KUKA KRL program: MyProgram_288().src

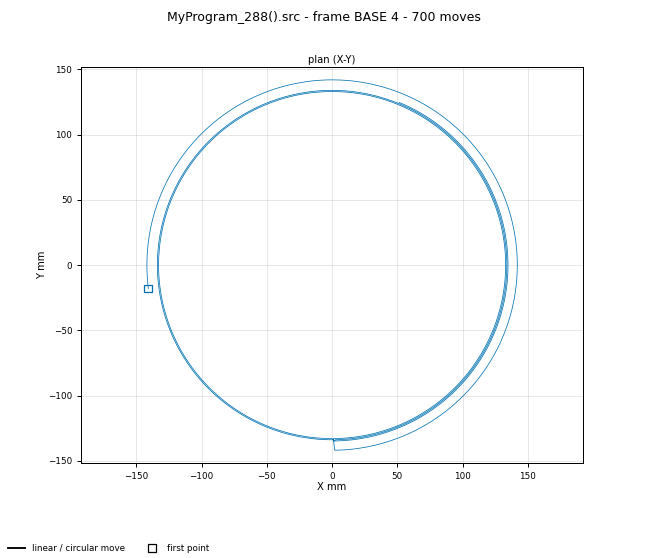
[picture p0: tool path of MyProgram_288().src in frame BASE 4, 700 of 700 moves have a stored position in this frame; points joined in program order, loops and branches not executed]
&ACCESS RVP
&REL 1
&PARAM TEMPLATE = C:\KRC\Roboter\Template\vorgabe
&PARAM EDITMASK = *
DEF MyProgram_288()
; ---- Setting reference (Base) ----
$BASE = BASE_DATA[4]

; --------------------------
; ---- Setting tool (TCP) ----
$TOOL = TOOL_DATA[3]
; --------------------------

$VEL.CP = VEL_APROX_PRINT
Startdeposition()
$VEL.CP = VEL_PRINT
LIN {X -140.7234,Y -17.946,Z 175,A -170.729,B 7.332,C 0.3003,E1 7.1791,E2 262.9088} C_DIS
LIN {X -141.1414,Y -14.3037,Z 175,A -172.2619,B 7.332,C 0.2967,E1 7.1786,E2 264.4473} C_DIS
LIN {X -141.4779,Y -10.4373,Z 175,A -173.8413,B 7.3323,C 0.2924,E1 7.1783,E2 266.0269} C_DIS
LIN {X -141.6907,Y -6.9788,Z 175,A -175.2622,B 7.3324,C 0.2887,E1 7.178,E2 267.4494} C_DIS
LIN {X -141.8124,Y -3.7701,Z 175,A -176.5843,B 7.3326,C 0.2853,E1 7.178,E2 268.7736} C_DIS
LIN {X -141.8652,Y -0.0247,Z 175,A -178.1224,B 7.3327,C 0.2813,E1 7.1779,E2 270.3138} C_DIS
LIN {X -141.8205,Y 3.4801,Z 175,A -179.5927,B 7.3328,C 0.2779,E1 7.1779,E2 271.7898} C_DIS
LIN {X -141.7054,Y 6.6857,Z 175,A 179.0865,B 7.333,C 0.2746,E1 7.1781,E2 273.1128} C_DIS
LIN {X -141.499,Y 10.1492,Z 175,A 177.6636,B 7.333,C 0.2708,E1 7.1784,E2 274.5373} C_DIS
LIN {X -141.1833,Y 13.8665,Z 175,A 176.1372,B 7.3332,C 0.2668,E1 7.1788,E2 276.0648} C_DIS
LIN {X -140.7964,Y 17.3669,Z 175,A 174.6904,B 7.3334,C 0.263,E1 7.1792,E2 277.5136} C_DIS
LIN {X -140.3316,Y 20.7961,Z 175,A 173.2648,B 7.3335,C 0.2594,E1 7.1798,E2 278.9414} C_DIS
LIN {X -139.825,Y 23.9636,Z 175,A 171.9397,B 7.3336,C 0.2561,E1 7.1804,E2 280.2692} C_DIS
LIN {X -139.1474,Y 27.6283,Z 175,A 170.388,B 7.3337,C 0.2525,E1 7.1812,E2 281.8255} C_DIS
LIN {X -138.5463,Y 30.4976,Z 175,A 169.1448,B 7.3338,C 0.2499,E1 7.1819,E2 283.0752} C_DIS
LIN {X -137.6088,Y 34.4796,Z 175,A 167.4991,B 7.334,C 0.2452,E1 7.183,E2 284.7185} C_DIS
LIN {X -136.7221,Y 37.8424,Z 175,A 166.1483,B 7.3341,C 0.2406,E1 7.184,E2 286.061} C_DIS
LIN {X -135.8307,Y 40.9296,Z 175,A 164.745,B 7.3342,C 0.2384,E1 7.1851,E2 287.4766} C_DIS
LIN {X -134.7033,Y 44.4966,Z 175,A 163.206,B 7.3343,C 0.2346,E1 7.1864,E2 289.0178} C_DIS
LIN {X -133.6609,Y 47.5391,Z 175,A 161.8116,B 7.3344,C 0.2324,E1 7.1877,E2 290.4232} C_DIS
LIN {X -132.3609,Y 51.0445,Z 175,A 160.4261,B 7.3346,C 0.2266,E1 7.1891,E2 291.7913} C_DIS
LIN {X -131.2247,Y 53.9034,Z 175,A 159.0704,B 7.3346,C 0.2248,E1 7.1905,E2 293.1604} C_DIS
LIN {X -129.8606,Y 57.112,Z 175,A 157.5842,B 7.3347,C 0.2221,E1 7.1922,E2 294.6552} C_DIS
LIN {X -128.3684,Y 60.3909,Z 175,A 156.1693,B 7.3349,C 0.2178,E1 7.1938,E2 296.0636} C_DIS
LIN {X -127.1018,Y 63.008,Z 175,A 154.9452,B 7.3349,C 0.2154,E1 7.1953,E2 297.2929} C_DIS
LIN {X -125.1762,Y 66.7568,Z 175,A 153.2018,B 7.335,C 0.2116,E1 7.1976,E2 299.04} C_DIS
LIN {X -123.1184,Y 70.4789,Z 175,A 151.466,B 7.3351,C 0.2075,E1 7.2,E2 300.7764} C_DIS
LIN {X -121.2352,Y 73.6715,Z 175,A 149.9398,B 7.3352,C 0.2042,E1 7.2021,E2 302.3049} C_DIS
LIN {X -118.9968,Y 77.2342,Z 175,A 148.2034,B 7.3353,C 0.2006,E1 7.2048,E2 304.0443} C_DIS
LIN {X -117.0516,Y 80.1517,Z 175,A 146.7407,B 7.3354,C 0.1978,E1 7.207,E2 305.5116} C_DIS
LIN {X -114.4633,Y 83.8067,Z 175,A 144.8252,B 7.3354,C 0.195,E1 7.2102,E2 307.439} C_DIS
LIN {X -111.8255,Y 87.2959,Z 175,A 143.1344,B 7.3356,C 0.1899,E1 7.213,E2 309.1185} C_DIS
LIN {X -109.1286,Y 90.6441,Z 175,A 141.2584,B 7.3356,C 0.188,E1 7.2164,E2 311.0106} C_DIS
LIN {X -106.2303,Y 94.0238,Z 175,A 139.4357,B 7.3358,C 0.1844,E1 7.2197,E2 312.8347} C_DIS
LIN {X -102.8784,Y 97.6811,Z 175,A 137.4601,B 7.3358,C 0.1798,E1 7.2235,E2 314.8049} C_DIS
LIN {X -99.7959,Y 100.8276,Z 175,A 135.6913,B 7.336,C 0.176,E1 7.227,E2 316.5708} C_DIS
LIN {X -96.667,Y 103.8308,Z 175,A 133.9289,B 7.336,C 0.1726,E1 7.2305,E2 318.3329} C_DIS
LIN {X -93.4431,Y 106.7417,Z 175,A 132.149,B 7.3361,C 0.1696,E1 7.2342,E2 320.1146} C_DIS
LIN {X -90.672,Y 109.1055,Z 175,A 130.5573,B 7.3361,C 0.1686,E1 7.2377,E2 321.7203} C_DIS
LIN {X -87.4029,Y 111.7415,Z 175,A 128.9292,B 7.3362,C 0.1646,E1 7.2412,E2 323.3382} C_DIS
LIN {X -83.8422,Y 114.4372,Z 175,A 127.0041,B 7.3362,C 0.1632,E1 7.2456,E2 325.2771} C_DIS
LIN {X -80.1816,Y 117.0311,Z 175,A 125.1904,B 7.3363,C 0.1603,E1 7.2497,E2 327.0895} C_DIS
LIN {X -76.6264,Y 119.3892,Z 175,A 123.4418,B 7.3363,C 0.1579,E1 7.2538,E2 328.8399} C_DIS
LIN {X -72.8225,Y 121.7468,Z 175,A 121.6324,B 7.3364,C 0.1553,E1 7.2581,E2 330.648} C_DIS
LIN {X -69.0599,Y 123.9203,Z 175,A 119.8443,B 7.3364,C 0.1532,E1 7.2625,E2 332.439} C_DIS
LIN {X -65.3363,Y 125.9223,Z 175,A 118.2406,B 7.3366,C 0.1494,E1 7.2664,E2 334.0281} C_DIS
LIN {X -62.3478,Y 127.4274,Z 175,A 116.9025,B 7.3366,C 0.1475,E1 7.2697,E2 335.3635} C_DIS
LIN {X -59.0667,Y 128.9814,Z 175,A 115.3957,B 7.3366,C 0.1463,E1 7.2736,E2 336.8742} C_DIS
LIN {X -55.8949,Y 130.3869,Z 175,A 113.9847,B 7.3366,C 0.1448,E1 7.2772,E2 338.2854} C_DIS
LIN {X -52.6901,Y 131.7145,Z 175,A 112.5741,B 7.3366,C 0.1434,E1 7.2808,E2 339.6962} C_DIS
LIN {X -49.6954,Y 132.8728,Z 175,A 111.2695,B 7.3366,C 0.1422,E1 7.2842,E2 341.0008} C_DIS
LIN {X -46.1824,Y 134.1346,Z 175,A 109.8377,B 7.3367,C 0.1396,E1 7.288,E2 342.422} C_DIS
LIN {X -43.0961,Y 135.1575,Z 175,A 108.3928,B 7.3367,C 0.1405,E1 7.2919,E2 343.8827} C_DIS
LIN {X -39.5162,Y 136.2477,Z 175,A 106.9116,B 7.3367,C 0.1388,E1 7.2958,E2 345.3591} C_DIS
LIN {X -36.4172,Y 137.1082,Z 175,A 105.7185,B 7.3368,C 0.1362,E1 7.299,E2 346.5378} C_DIS
LIN {X -33.032,Y 137.963,Z 175,A 104.1617,B 7.3368,C 0.1375,E1 7.3033,E2 348.1124} C_DIS
LIN {X -29.4095,Y 138.7812,Z 175,A 102.7067,B 7.3368,C 0.1359,E1 7.3072,E2 349.5608} C_DIS
LIN {X -26.2675,Y 139.4096,Z 175,A 101.3667,B 7.3368,C 0.1359,E1 7.3109,E2 350.9058} C_DIS
LIN {X -22.5864,Y 140.0547,Z 175,A 99.8841,B 7.3368,C 0.1347,E1 7.315,E2 352.3841} C_DIS
LIN {X -19.3533,Y 140.5378,Z 175,A 98.557,B 7.3368,C 0.1343,E1 7.3186,E2 353.7114} C_DIS
LIN {X -15.9024,Y 140.97,Z 175,A 97.1856,B 7.3368,C 0.1333,E1 7.3224,E2 355.0778} C_DIS
LIN {X -12.4434,Y 141.3164,Z 175,A 95.6611,B 7.3368,C 0.1348,E1 7.3267,E2 356.6168} C_DIS
LIN {X -8.7043,Y 141.5951,Z 175,A 94.091,B 7.3368,C 0.1354,E1 7.3311,E2 358.1931} C_DIS
LIN {X -3.7458,Y 141.8131,Z 175,A 92.2151,B 7.3368,C 0.1332,E1 7.3363,E2 360.0518} C_DIS
LIN {X -0.0049,Y 141.8646,Z 175,A 90.7261,B 7.3368,C 0.1328,E1 7.3404,E2 361.5374} C_DIS
LIN {X 3.4708,Y 141.8207,Z 175,A 89.2787,B 7.3368,C 0.1336,E1 7.3445,E2 362.9897} C_DIS
LIN {X 6.6856,Y 141.7054,Z 175,A 88.1474,B 7.3369,C 0.131,E1 7.3476,E2 364.0991} C_DIS
LIN {X 10.1728,Y 141.4972,Z 175,A 86.5809,B 7.3369,C 0.1338,E1 7.352,E2 365.6848} C_DIS
LIN {X 13.8225,Y 141.1876,Z 175,A 85.1063,B 7.3369,C 0.1341,E1 7.3561,E2 367.1583} C_DIS
LIN {X 17.3556,Y 140.7977,Z 175,A 83.6862,B 7.3369,C 0.1343,E1 7.36,E2 368.5759} C_DIS
LIN {X 20.8036,Y 140.3305,Z 175,A 82.2883,B 7.3369,C 0.1348,E1 7.3639,E2 369.9724} C_DIS
LIN {X 23.9936,Y 139.82,Z 175,A 80.9825,B 7.3369,C 0.1354,E1 7.3675,E2 371.278} C_DIS
LIN {X 27.669,Y 139.1391,Z 175,A 79.4623,B 7.3369,C 0.1364,E1 7.3717,E2 372.7991} C_DIS
LIN {X 30.8166,Y 138.4768,Z 175,A 78.1663,B 7.3368,C 0.1372,E1 7.3752,E2 374.0944} C_DIS
LIN {X 34.4536,Y 137.6154,Z 175,A 76.678,B 7.3368,C 0.1378,E1 7.3792,E2 375.5795} C_DIS
LIN {X 37.5658,Y 136.7995,Z 175,A 75.3703,B 7.3368,C 0.1389,E1 7.3828,E2 376.8881} C_DIS
LIN {X 40.9301,Y 135.8305,Z 175,A 73.9723,B 7.3368,C 0.1398,E1 7.3865,E2 378.2837} C_DIS
LIN {X 44.4992,Y 134.7025,Z 175,A 72.471,B 7.3368,C 0.1409,E1 7.3905,E2 379.7834} C_DIS
LIN {X 47.5418,Y 133.6599,Z 175,A 71.1119,B 7.3367,C 0.1432,E1 7.3941,E2 381.15} C_DIS
LIN {X 50.7421,Y 132.4785,Z 175,A 69.7924,B 7.3367,C 0.1436,E1 7.3975,E2 382.462} C_DIS
LIN {X 54.0426,Y 131.1665,Z 175,A 68.4561,B 7.3367,C 0.1434,E1 7.4009,E2 383.7856} C_DIS
LIN {X 57.2208,Y 129.812,Z 175,A 67.0402,B 7.3367,C 0.1454,E1 7.4046,E2 385.204} C_DIS
LIN {X 60.5278,Y 128.303,Z 175,A 65.5555,B 7.3366,C 0.1475,E1 7.4084,E2 386.6908} C_DIS
LIN {X 63.7676,Y 126.7238,Z 175,A 64.1131,B 7.3366,C 0.1491,E1 7.412,E2 388.1315} C_DIS
LIN {X 66.972,Y 125.0606,Z 175,A 62.5572,B 7.3365,C 0.1528,E1 7.4158,E2 389.6998} C_DIS
LIN {X 70.5636,Y 123.0701,Z 175,A 61.0143,B 7.3365,C 0.153,E1 7.4196,E2 391.2281} C_DIS
LIN {X 73.6814,Y 121.2291,Z 175,A 59.5513,B 7.3365,C 0.1552,E1 7.4231,E2 392.6911} C_DIS
LIN {X 77.2493,Y 118.987,Z 175,A 57.8432,B 7.3364,C 0.1579,E1 7.4271,E2 394.4002} C_DIS
LIN {X 80.8578,Y 116.565,Z 175,A 56.1235,B 7.3364,C 0.1601,E1 7.431,E2 396.1156} C_DIS
LIN {X 83.9138,Y 114.3846,Z 175,A 54.5575,B 7.3363,C 0.1636,E1 7.4346,E2 397.6881} C_DIS
LIN {X 87.2776,Y 111.84,Z 175,A 52.9629,B 7.3363,C 0.1646,E1 7.4381,E2 399.269} C_DIS
LIN {X 90.0964,Y 109.5818,Z 175,A 51.4076,B 7.3361,C 0.169,E1 7.4415,E2 400.837} C_DIS
LIN {X 93.4073,Y 106.7729,Z 175,A 49.6713,B 7.3361,C 0.1719,E1 7.4452,E2 402.5715} C_DIS
LIN {X 96.6022,Y 103.8911,Z 175,A 47.9865,B 7.3361,C 0.1743,E1 7.4486,E2 404.2499} C_DIS
LIN {X 99.7897,Y 100.8337,Z 175,A 46.2137,B 7.3359,C 0.1777,E1 7.4522,E2 406.0217} C_DIS
LIN {X 102.8319,Y 97.7298,Z 175,A 44.4517,B 7.3359,C 0.1814,E1 7.4556,E2 407.7852} C_DIS
LIN {X 106.1796,Y 94.0812,Z 175,A 42.5729,B 7.3358,C 0.1834,E1 7.4591,E2 409.6491} C_DIS
LIN {X 109.0702,Y 90.7146,Z 175,A 40.7283,B 7.3357,C 0.1883,E1 7.4624,E2 411.501} C_DIS
LIN {X 111.7052,Y 87.4492,Z 175,A 39.1485,B 7.3357,C 0.1899,E1 7.4651,E2 413.0667} C_DIS
LIN {X 114.3842,Y 83.9144,Z 175,A 37.3384,B 7.3355,C 0.1944,E1 7.4682,E2 414.8799} C_DIS
LIN {X 116.9834,Y 80.2511,Z 175,A 35.5118,B 7.3354,C 0.1989,E1 7.4711,E2 416.7089} C_DIS
LIN {X 119.3861,Y 76.6312,Z 175,A 33.7922,B 7.3353,C 0.2024,E1 7.4737,E2 418.4249} C_DIS
LIN {X 121.7449,Y 72.8257,Z 175,A 32.0304,B 7.3352,C 0.2059,E1 7.4763,E2 420.1816} C_DIS
LIN {X 123.9194,Y 69.0615,Z 175,A 30.289,B 7.3351,C 0.21,E1 7.4787,E2 421.922} C_DIS
LIN {X 125.9235,Y 65.3341,Z 175,A 28.726,B 7.3351,C 0.2115,E1 7.4807,E2 423.467} C_DIS
LIN {X 127.4362,Y 62.3301,Z 175,A 27.3886,B 7.3349,C 0.2146,E1 7.4823,E2 424.8024} C_DIS
LIN {X 128.8558,Y 59.3382,Z 175,A 26.0433,B 7.3349,C 0.2182,E1 7.4839,E2 426.1495} C_DIS
LIN {X 130.3837,Y 55.9023,Z 175,A 24.5848,B 7.3348,C 0.221,E1 7.4855,E2 427.601} C_DIS
LIN {X 132.0043,Y 51.9619,Z 175,A 22.7479,B 7.3345,C 0.2279,E1 7.4875,E2 429.4541} C_DIS
LIN {X 133.4807,Y 48.0388,Z 175,A 21.1983,B 7.3345,C 0.2296,E1 7.489,E2 430.9862} C_DIS
LIN {X 134.6186,Y 44.7511,Z 175,A 19.8558,B 7.3345,C 0.2322,E1 7.4902,E2 432.3215} C_DIS
LIN {X 135.7526,Y 41.1849,Z 175,A 18.3369,B 7.3343,C 0.2365,E1 7.4914,E2 433.8424} C_DIS
LIN {X 137.036,Y 36.6878,Z 175,A 16.4669,B 7.3341,C 0.2413,E1 7.4928,E2 435.7112} C_DIS
LIN {X 137.9658,Y 33.0204,Z 175,A 14.9942,B 7.3341,C 0.2445,E1 7.4938,E2 437.1779} C_DIS
LIN {X 138.789,Y 29.3734,Z 175,A 13.5616,B 7.3339,C 0.2472,E1 7.4946,E2 438.6015} C_DIS
LIN {X 139.4177,Y 26.225,Z 175,A 12.2541,B 7.3338,C 0.2511,E1 7.4953,E2 439.9114} C_DIS
LIN {X 140.0621,Y 22.5423,Z 175,A 10.8004,B 7.3337,C 0.2543,E1 7.496,E2 441.359} C_DIS
LIN {X 140.5364,Y 19.363,Z 175,A 9.5261,B 7.3336,C 0.2575,E1 7.4965,E2 442.6311} C_DIS
LIN {X 140.969,Y 15.9119,Z 175,A 8.1148,B 7.3334,C 0.2616,E1 7.497,E2 444.0444} C_DIS
LIN {X 141.3173,Y 12.4337,Z 175,A 6.6844,B 7.3333,C 0.266,E1 7.4974,E2 445.4784} C_DIS
LIN {X 141.5951,Y 8.7044,Z 175,A 5.2719,B 7.3332,C 0.2684,E1 7.4976,E2 446.8792} C_DIS
LIN {X 141.7662,Y 5.2318,Z 175,A 3.9319,B 7.3331,C 0.2712,E1 7.4978,E2 448.212} C_DIS
LIN {X 141.8423,Y 2.388,Z 175,A 2.8266,B 7.333,C 0.2736,E1 7.4978,E2 449.3126} C_DIS
LIN {X 141.8603,Y -0.9287,Z 175,A 1.3827,B 7.3328,C 0.2795,E1 7.4978,E2 450.7714} C_DIS
LIN {X 141.7668,Y -5.2171,Z 175,A -0.1909,B 7.3328,C 0.2814,E1 7.4978,E2 452.3256} C_DIS
LIN {X 141.6121,Y -8.4285,Z 175,A -1.5263,B 7.3325,C 0.2858,E1 7.4975,E2 453.667} C_DIS
LIN {X 141.3626,Y -11.897,Z 175,A -2.936,B 7.3324,C 0.29,E1 7.4972,E2 455.0787} C_DIS
LIN {X 140.9984,Y -15.6386,Z 175,A -4.3756,B 7.3323,C 0.2928,E1 7.4968,E2 456.5093} C_DIS
LIN {X 140.5736,Y -19.089,Z 175,A -5.7505,B 7.3321,C 0.2962,E1 7.4963,E2 457.8817} C_DIS
LIN {X 140.0642,Y -22.5294,Z 175,A -7.124,B 7.332,C 0.2996,E1 7.4957,E2 459.2524} C_DIS
LIN {X 139.5169,Y -25.6986,Z 175,A -8.4695,B 7.3318,C 0.3042,E1 7.4951,E2 460.6052} C_DIS
LIN {X 138.7863,Y -29.3861,Z 175,A -9.7964,B 7.3318,C 0.3047,E1 7.4944,E2 461.9083} C_DIS
LIN {X 138.0874,Y -32.5157,Z 175,A -11.2484,B 7.3315,C 0.3115,E1 7.4934,E2 463.3822} C_DIS
LIN {X 137.3528,Y -35.4882,Z 175,A -12.5164,B 7.3313,C 0.3156,E1 7.4926,E2 464.6555} C_DIS
LIN {X 136.3305,Y -39.2334,Z 175,A -13.9267,B 7.3313,C 0.3169,E1 7.4915,E2 466.0465} C_DIS
LIN {X 135.3282,Y -42.5618,Z 175,A -15.3792,B 7.3311,C 0.3217,E1 7.4903,E2 467.5068} C_DIS
LIN {X 134.1473,Y -46.1459,Z 175,A -16.7226,B 7.3311,C 0.3223,E1 7.4891,E2 468.8278} C_DIS
LIN {X 132.9692,Y -49.4381,Z 175,A -18.1829,B 7.3308,C 0.3271,E1 7.4877,E2 470.2958} C_DIS
LIN {X 131.9432,Y -52.1189,Z 175,A -19.3932,B 7.3306,C 0.3313,E1 7.4865,E2 471.514} C_DIS
LIN {X 130.4934,Y -55.6486,Z 175,A -20.8303,B 7.3306,C 0.3334,E1 7.485,E2 472.9389} C_DIS
LIN {X 129.3945,Y -58.1542,Z 175,A -21.9769,B 7.3304,C 0.3371,E1 7.4836,E2 474.092} C_DIS
LIN {X 127.5676,Y -62.0635,Z 175,A -23.6711,B 7.3302,C 0.3408,E1 7.4816,E2 475.7815} C_DIS
LIN {X 125.9439,Y -65.2952,Z 175,A -25.0621,B 7.3301,C 0.3432,E1 7.4799,E2 477.1648} C_DIS
LIN {X 123.9234,Y -69.0543,Z 175,A -26.8101,B 7.3299,C 0.3481,E1 7.4775,E2 478.9177} C_DIS
LIN {X 121.7489,Y -72.819,Z 175,A -28.5238,B 7.3297,C 0.3517,E1 7.4751,E2 480.6275} C_DIS
LIN {X 119.3813,Y -76.6388,Z 175,A -30.2905,B 7.3295,C 0.3553,E1 7.4725,E2 482.3895} C_DIS
LIN {X 117.0597,Y -80.14,Z 175,A -31.9621,B 7.3293,C 0.3589,E1 7.4699,E2 484.0595} C_DIS
LIN {X 114.9118,Y -83.1904,Z 175,A -33.5419,B 7.3291,C 0.364,E1 7.4673,E2 485.6505} C_DIS
LIN {X 112.3925,Y -86.5648,Z 175,A -35.1214,B 7.3291,C 0.3656,E1 7.4647,E2 487.2155} C_DIS
LIN {X 109.7464,Y -89.895,Z 175,A -36.8076,B 7.3288,C 0.369,E1 7.4617,E2 488.8992} C_DIS
LIN {X 107.3387,Y -92.7567,Z 175,A -38.4061,B 7.3286,C 0.3741,E1 7.4588,E2 490.5108} C_DIS
LIN {X 104.0357,Y -96.447,Z 175,A -40.3522,B 7.3284,C 0.3774,E1 7.4551,E2 492.4517} C_DIS
LIN {X 100.8336,Y -99.7899,Z 175,A -42.1942,B 7.3282,C 0.3809,E1 7.4516,E2 494.2917} C_DIS
LIN {X 97.7289,Y -102.8327,Z 175,A -43.9565,B 7.328,C 0.3846,E1 7.448,E2 496.0566} C_DIS
LIN {X 94.0795,Y -106.1811,Z 175,A -45.8383,B 7.328,C 0.3864,E1 7.4441,E2 497.9245} C_DIS
LIN {X 90.6676,Y -109.1091,Z 175,A -47.7043,B 7.3277,C 0.3909,E1 7.4401,E2 499.7988} C_DIS
LIN {X 87.3868,Y -111.7542,Z 175,A -49.3003,B 7.3277,C 0.392,E1 7.4367,E2 501.3822} C_DIS
LIN {X 83.8166,Y -114.456,Z 175,A -51.1809,B 7.3274,C 0.3967,E1 7.4324,E2 503.2741} C_DIS
LIN {X 80.2558,Y -116.9802,Z 175,A -52.9136,B 7.3273,C 0.3992,E1 7.4285,E2 505.0043} C_DIS
LIN {X 76.6377,Y -119.382,Z 175,A -54.6428,B 7.3271,C 0.4016,E1 7.4244,E2 506.7317} C_DIS
LIN {X 72.8366,Y -121.7384,Z 175,A -56.4145,B 7.3271,C 0.4038,E1 7.4202,E2 508.5004} C_DIS
LIN {X 69.0737,Y -123.9126,Z 175,A -58.1684,B 7.3269,C 0.4065,E1 7.416,E2 510.2556} C_DIS
LIN {X 65.3342,Y -125.9234,Z 175,A -59.7466,B 7.3269,C 0.4065,E1 7.4121,E2 511.817} C_DIS
LIN {X 62.3344,Y -127.434,Z 175,A -61.0925,B 7.3268,C 0.4081,E1 7.4087,E2 513.1625} C_DIS
LIN {X 59.0848,Y -128.973,Z 175,A -62.5312,B 7.3267,C 0.4098,E1 7.4051,E2 514.6006} C_DIS
LIN {X 55.9173,Y -130.3773,Z 175,A -63.9205,B 7.3266,C 0.4114,E1 7.4015,E2 515.9896} C_DIS
LIN {X 52.6788,Y -131.719,Z 175,A -65.2318,B 7.3266,C 0.4111,E1 7.3982,E2 517.288} C_DIS
LIN {X 49.6815,Y -132.878,Z 175,A -66.6073,B 7.3264,C 0.414,E1 7.3946,E2 518.6748} C_DIS
LIN {X 46.1632,Y -134.1413,Z 175,A -68.0719,B 7.3264,C 0.4148,E1 7.3907,E2 520.1346} C_DIS
LIN {X 43.1102,Y -135.153,Z 175,A -69.4357,B 7.3263,C 0.4173,E1 7.3871,E2 521.5079} C_DIS
LIN {X 39.5137,Y -136.2484,Z 175,A -70.8199,B 7.3263,C 0.4163,E1 7.3834,E2 522.8752} C_DIS
LIN {X 36.3953,Y -137.114,Z 175,A -72.2029,B 7.3262,C 0.4188,E1 7.3797,E2 524.2693} C_DIS
LIN {X 33.0274,Y -137.9641,Z 175,A -73.6256,B 7.3261,C 0.4203,E1 7.3758,E2 525.6956} C_DIS
LIN {X 29.3832,Y -138.7869,Z 175,A -75.0769,B 7.3261,C 0.4203,E1 7.3718,E2 527.1401} C_DIS
LIN {X 26.4252,Y -139.3794,Z 175,A -76.3544,B 7.326,C 0.4222,E1 7.3683,E2 528.4262} C_DIS
LIN {X 22.5515,Y -140.0606,Z 175,A -77.8805,B 7.326,C 0.4221,E1 7.3641,E2 529.9451} C_DIS
LIN {X 19.3702,Y -140.5354,Z 175,A -79.176,B 7.326,C 0.4227,E1 7.3605,E2 531.2409} C_DIS
LIN {X 15.899,Y -140.9704,Z 175,A -80.6133,B 7.3259,C 0.4238,E1 7.3566,E2 532.6823} C_DIS
LIN {X 12.4382,Y -141.3169,Z 175,A -82.0666,B 7.3259,C 0.4251,E1 7.3525,E2 534.1427} C_DIS
LIN {X 8.7096,Y -141.5948,Z 175,A -83.5038,B 7.3259,C 0.4244,E1 7.3485,E2 535.571} C_DIS
LIN {X 5.226,Y -141.7664,Z 175,A -84.8723,B 7.3259,C 0.424,E1 7.3447,E2 536.9349} C_DIS
LIN {X 2.0041,Y -141.8487,Z 175,A -86.2176,B 7.3259,C 0.425,E1 7.3409,E2 538.2867} C_DIS
LIN {X 2.0041,Y -141.8487,Z 175,A -86.2176,B 7.3259,C 0.425,E1 7.3409,E2 538.2867} C_DIS
Enddeposition()
LIN {X 0.9626,Y -132.9228,Z 176,A -86.6434,B 7.2072,C 0.3831,E1 7.2198,E2 538.4124} C_DIS
Startdeposition()
$VEL.CP = VEL_PRINT
LIN {X 3.2583,Y -132.8887,Z 176,A -85.2667,B 7.2075,C 0.3768,E1 7.2238,E2 536.9873} C_DIS
LIN {X 6.5134,Y -132.7684,Z 176,A -83.7452,B 7.2077,C 0.3746,E1 7.2281,E2 535.4504} C_DIS
LIN {X 10.6957,Y -132.4978,Z 176,A -81.8954,B 7.2077,C 0.3733,E1 7.2332,E2 533.5942} C_DIS
LIN {X 14.6526,Y -132.1185,Z 176,A -80.2271,B 7.2077,C 0.3733,E1 7.2379,E2 531.9306} C_DIS
LIN {X 18.5813,Y -131.6229,Z 176,A -78.584,B 7.2077,C 0.3735,E1 7.2424,E2 530.2944} C_DIS
LIN {X 22.0161,Y -131.0919,Z 176,A -77.18,B 7.2077,C 0.3742,E1 7.2462,E2 528.9013} C_DIS
LIN {X 25.2184,Y -130.5139,Z 176,A -75.7465,B 7.2077,C 0.3727,E1 7.2502,E2 527.4631} C_DIS
LIN {X 29.1223,Y -129.6993,Z 176,A -74.0293,B 7.2078,C 0.3715,E1 7.2549,E2 525.745} C_DIS
LIN {X 32.9748,Y -128.773,Z 176,A -72.3144,B 7.2078,C 0.37,E1 7.2595,E2 524.0281} C_DIS
LIN {X 36.3332,Y -127.8669,Z 176,A -70.8628,B 7.2079,C 0.3695,E1 7.2634,E2 522.5814} C_DIS
LIN {X 39.4727,Y -126.933,Z 176,A -69.2854,B 7.2081,C 0.3654,E1 7.2677,E2 520.9823} C_DIS
LIN {X 44.1289,Y -125.3904,Z 176,A -67.3434,B 7.2081,C 0.3661,E1 7.2728,E2 519.0604} C_DIS
LIN {X 47.8424,Y -124.0199,Z 176,A -65.6531,B 7.2081,C 0.3645,E1 7.2772,E2 517.3708} C_DIS
LIN {X 51.0798,Y -122.7216,Z 176,A -64.0481,B 7.2083,C 0.3609,E1 7.2814,E2 515.7519} C_DIS
LIN {X 55.3485,Y -120.8573,Z 176,A -62.021,B 7.2085,C 0.358,E1 7.2866,E2 513.7209} C_DIS
LIN {X 58.9228,Y -119.1546,Z 176,A -60.4468,B 7.2085,C 0.358,E1 7.2905,E2 512.1619} C_DIS
LIN {X 61.9888,Y -117.5888,Z 176,A -59.0729,B 7.2085,C 0.3577,E1 7.2939,E2 510.8004} C_DIS
LIN {X 65.4628,Y -115.6936,Z 176,A -57.3229,B 7.2087,C 0.3545,E1 7.2981,E2 509.0436} C_DIS
LIN {X 68.2015,Y -114.1,Z 176,A -55.871,B 7.2088,C 0.3508,E1 7.3017,E2 507.5798} C_DIS
LIN {X 71.8872,Y -111.8147,Z 176,A -54.1397,B 7.2088,C 0.3502,E1 7.3057,E2 505.8642} C_DIS
LIN {X 74.6185,Y -110.0106,Z 176,A -52.5968,B 7.2091,C 0.3455,E1 7.3093,E2 504.3035} C_DIS
LIN {X 78.4447,Y -107.3161,Z 176,A -50.7118,B 7.2091,C 0.3443,E1 7.3136,E2 502.4332} C_DIS
LIN {X 81.3997,Y -105.092,Z 176,A -49.0888,B 7.2093,C 0.3408,E1 7.3172,E2 500.8053} C_DIS
LIN {X 84.6009,Y -102.5328,Z 176,A -47.3309,B 7.2095,C 0.3376,E1 7.321,E2 499.0469} C_DIS
LIN {X 87.7841,Y -99.8213,Z 176,A -45.5136,B 7.2096,C 0.3338,E1 7.3248,E2 497.2261} C_DIS
LIN {X 91.0724,Y -96.8302,Z 176,A -43.6664,B 7.2098,C 0.3312,E1 7.3286,E2 495.3857} C_DIS
LIN {X 93.9956,Y -93.9959,Z 176,A -41.9441,B 7.2099,C 0.3281,E1 7.332,E2 493.6658} C_DIS
LIN {X 96.8298,Y -91.0728,Z 176,A -40.2137,B 7.2101,C 0.3247,E1 7.3354,E2 491.9367} C_DIS
LIN {X 99.5865,Y -88.0498,Z 176,A -38.4999,B 7.2101,C 0.3217,E1 7.3386,E2 490.2275} C_DIS
LIN {X 102.2373,Y -84.9577,Z 176,A -36.761,B 7.2104,C 0.3181,E1 7.3417,E2 488.489} C_DIS
LIN {X 104.7921,Y -81.7863,Z 176,A -34.9618,B 7.2106,C 0.3132,E1 7.3448,E2 486.6827} C_DIS
LIN {X 107.3182,Y -78.4419,Z 176,A -33.1894,B 7.2107,C 0.3096,E1 7.3478,E2 484.9128} C_DIS
LIN {X 109.9904,Y -74.6482,Z 176,A -31.294,B 7.2108,C 0.3066,E1 7.3508,E2 483.0285} C_DIS
LIN {X 112.3043,Y -71.1196,Z 176,A -29.5754,B 7.211,C 0.304,E1 7.3533,E2 481.3206} C_DIS
LIN {X 114.3788,Y -67.7338,Z 176,A -27.8469,B 7.2112,C 0.2994,E1 7.3558,E2 479.5883} C_DIS
LIN {X 116.1288,Y -64.6873,Z 176,A -26.274,B 7.2114,C 0.2944,E1 7.358,E2 478.0067} C_DIS
LIN {X 118.311,Y -60.5995,Z 176,A -24.3959,B 7.2114,C 0.2914,E1 7.3604,E2 476.1414} C_DIS
LIN {X 119.8469,Y -57.5018,Z 176,A -22.9863,B 7.2116,C 0.289,E1 7.3621,E2 474.7403} C_DIS
LIN {X 121.501,Y -53.92,Z 176,A -21.3103,B 7.2117,C 0.2849,E1 7.3641,E2 473.0657} C_DIS
LIN {X 122.6992,Y -51.1334,Z 176,A -19.9865,B 7.2119,C 0.2811,E1 7.3655,E2 471.7386} C_DIS
LIN {X 124.0192,Y -47.8443,Z 176,A -18.5281,B 7.2119,C 0.2783,E1 7.367,E2 470.2873} C_DIS
LIN {X 125.3898,Y -44.1306,Z 176,A -16.7909,B 7.2122,C 0.273,E1 7.3687,E2 468.5447} C_DIS
LIN {X 126.7228,Y -40.1395,Z 176,A -15.0786,B 7.2123,C 0.2699,E1 7.3701,E2 466.8431} C_DIS
LIN {X 127.6603,Y -37.0498,Z 176,A -13.715,B 7.2124,C 0.2666,E1 7.3712,E2 465.4817} C_DIS
LIN {X 128.5184,Y -33.9538,Z 176,A -12.3606,B 7.2126,C 0.2632,E1 7.3722,E2 464.1297} C_DIS
LIN {X 129.4237,Y -30.3289,Z 176,A -10.6299,B 7.2128,C 0.2565,E1 7.3733,E2 462.3828} C_DIS
LIN {X 130.3743,Y -25.9356,Z 176,A -8.8828,B 7.2128,C 0.2545,E1 7.3743,E2 460.6573} C_DIS
LIN {X 130.9712,Y -22.7332,Z 176,A -7.5096,B 7.213,C 0.2511,E1 7.375,E2 459.2867} C_DIS
LIN {X 131.6223,Y -18.5854,Z 176,A -5.7303,B 7.2131,C 0.2465,E1 7.3757,E2 457.5094} C_DIS
LIN {X 132.1183,Y -14.6545,Z 176,A -4.0419,B 7.2133,C 0.242,E1 7.3763,E2 455.8219} C_DIS
LIN {X 132.4963,Y -10.7131,Z 176,A -2.364,B 7.2134,C 0.2376,E1 7.3767,E2 454.146} C_DIS
LIN {X 132.7315,Y -7.2465,Z 176,A -0.9556,B 7.2135,C 0.235,E1 7.3769,E2 452.7473} C_DIS
LIN {X 132.8691,Y -3.9636,Z 176,A 0.4838,B 7.2137,C 0.2305,E1 7.3771,E2 451.3039} C_DIS
LIN {X 132.9297,Y -0.2794,Z 176,A 2.1045,B 7.2138,C 0.2253,E1 7.3771,E2 449.6778} C_DIS
LIN {X 132.8889,Y 3.2543,Z 176,A 3.54,B 7.2139,C 0.2225,E1 7.3771,E2 448.2518} C_DIS
LIN {X 132.7685,Y 6.5105,Z 176,A 4.9117,B 7.214,C 0.2191,E1 7.3769,E2 446.8829} C_DIS
LIN {X 132.5677,Y 9.7794,Z 176,A 6.2834,B 7.2141,C 0.2158,E1 7.3766,E2 445.5149} C_DIS
LIN {X 132.2183,Y 13.7251,Z 176,A 8.0246,B 7.2143,C 0.2103,E1 7.3762,E2 443.7683} C_DIS
LIN {X 131.7215,Y 17.8778,Z 176,A 9.7158,B 7.2143,C 0.2072,E1 7.3756,E2 442.0893} C_DIS
LIN {X 131.2416,Y 21.119,Z 176,A 11.0953,B 7.2145,C 0.2038,E1 7.375,E2 440.7128} C_DIS
LIN {X 130.5103,Y 25.2374,Z 176,A 12.8769,B 7.2145,C 0.1991,E1 7.3741,E2 438.9323} C_DIS
LIN {X 129.7001,Y 29.1187,Z 176,A 14.7033,B 7.2148,C 0.1922,E1 7.373,E2 437.0905} C_DIS
LIN {X 128.7707,Y 32.9842,Z 176,A 16.2577,B 7.2148,C 0.1903,E1 7.372,E2 435.5542} C_DIS
LIN {X 127.8634,Y 36.3458,Z 176,A 17.8586,B 7.215,C 0.1843,E1 7.3708,E2 433.94} C_DIS
LIN {X 126.7162,Y 40.1599,Z 176,A 19.519,B 7.215,C 0.1807,E1 7.3694,E2 432.2854} C_DIS
LIN {X 125.4139,Y 44.0612,Z 176,A 21.1357,B 7.2151,C 0.1787,E1 7.3679,E2 430.6865} C_DIS
LIN {X 124.0313,Y 47.813,Z 176,A 22.8968,B 7.2153,C 0.1734,E1 7.3662,E2 428.9198} C_DIS
LIN {X 122.4551,Y 51.718,Z 176,A 24.6096,B 7.2153,C 0.1705,E1 7.3644,E2 427.2183} C_DIS
LIN {X 120.8543,Y 55.3548,Z 176,A 26.2827,B 7.2154,C 0.1667,E1 7.3625,E2 425.5491} C_DIS
LIN {X 119.4618,Y 58.3,Z 176,A 27.6604,B 7.2154,C 0.1636,E1 7.3608,E2 424.1737} C_DIS
LIN {X 118.0387,Y 61.132,Z 176,A 29.0202,B 7.2156,C 0.1602,E1 7.3591,E2 422.8141} C_DIS
LIN {X 116.4495,Y 64.1082,Z 176,A 30.57,B 7.2156,C 0.1548,E1 7.357,E2 421.2519} C_DIS
LIN {X 114.3753,Y 67.7397,Z 176,A 32.2047,B 7.2157,C 0.1534,E1 7.3547,E2 419.6366} C_DIS
LIN {X 112.6816,Y 70.5209,Z 176,A 33.5929,B 7.2157,C 0.1503,E1 7.3527,E2 418.2496} C_DIS
LIN {X 110.9187,Y 73.2618,Z 176,A 34.9712,B 7.2158,C 0.1474,E1 7.3506,E2 416.8739} C_DIS
LIN {X 108.6854,Y 76.5358,Z 176,A 36.7728,B 7.2159,C 0.1417,E1 7.3477,E2 415.0602} C_DIS
LIN {X 106.2211,Y 79.9208,Z 176,A 38.4714,B 7.2159,C 0.1394,E1 7.3449,E2 413.3738} C_DIS
LIN {X 103.816,Y 83.0215,Z 176,A 40.1481,B 7.2161,C 0.1359,E1 7.342,E2 411.6982} C_DIS
LIN {X 101.2748,Y 86.1025,Z 176,A 41.8889,B 7.2161,C 0.1318,E1 7.3389,E2 409.9544} C_DIS
LIN {X 98.4963,Y 89.2677,Z 176,A 43.6538,B 7.2161,C 0.1288,E1 7.3356,E2 408.1951} C_DIS
LIN {X 95.7047,Y 92.2546,Z 176,A 45.4042,B 7.2162,C 0.1253,E1 7.3322,E2 406.4456} C_DIS
LIN {X 92.8371,Y 95.14,Z 176,A 47.1714,B 7.2163,C 0.1216,E1 7.3287,E2 404.6762} C_DIS
LIN {X 89.5427,Y 98.2467,Z 176,A 49.0388,B 7.2163,C 0.1192,E1 7.3249,E2 402.8185} C_DIS
LIN {X 86.5802,Y 100.867,Z 176,A 50.7389,B 7.2164,C 0.1161,E1 7.3213,E2 401.1186} C_DIS
LIN {X 83.4271,Y 103.4898,Z 176,A 52.4645,B 7.2164,C 0.1136,E1 7.3176,E2 399.3978} C_DIS
LIN {X 79.9382,Y 106.208,Z 176,A 54.307,B 7.2164,C 0.1114,E1 7.3136,E2 397.5627} C_DIS
LIN {X 77.1404,Y 108.2572,Z 176,A 55.7511,B 7.2165,C 0.1097,E1 7.3103,E2 396.1244} C_DIS
LIN {X 73.9201,Y 110.4811,Z 176,A 57.4136,B 7.2165,C 0.1074,E1 7.3065,E2 394.4646} C_DIS
LIN {X 71.1184,Y 112.3051,Z 176,A 58.8416,B 7.2165,C 0.1054,E1 7.3031,E2 393.0382} C_DIS
LIN {X 67.7418,Y 114.374,Z 176,A 60.5789,B 7.2166,C 0.1024,E1 7.299,E2 391.2971} C_DIS
LIN {X 64.7288,Y 116.1058,Z 176,A 61.9909,B 7.2166,C 0.1017,E1 7.2956,E2 389.8954} C_DIS
LIN {X 62.0536,Y 117.5547,Z 176,A 63.316,B 7.2166,C 0.0997,E1 7.2923,E2 388.5685} C_DIS
LIN {X 58.9331,Y 119.1495,Z 176,A 64.8114,B 7.2166,C 0.0979,E1 7.2886,E2 387.075} C_DIS
LIN {X 55.9933,Y 120.5591,Z 176,A 66.328,B 7.2167,C 0.0944,E1 7.2847,E2 385.5452} C_DIS
LIN {X 52.3741,Y 122.1754,Z 176,A 68.0216,B 7.2167,C 0.0927,E1 7.2804,E2 383.8535} C_DIS
LIN {X 48.3452,Y 123.8245,Z 176,A 69.8598,B 7.2167,C 0.0913,E1 7.2756,E2 382.02} C_DIS
LIN {X 44.787,Y 125.1557,Z 176,A 71.3891,B 7.2167,C 0.0914,E1 7.2716,E2 380.5039} C_DIS
LIN {X 41.2342,Y 126.3729,Z 176,A 73.0617,B 7.2167,C 0.0891,E1 7.2672,E2 378.8252} C_DIS
LIN {X 37.055,Y 127.6588,Z 176,A 74.9684,B 7.2168,C 0.0872,E1 7.2621,E2 376.9162} C_DIS
LIN {X 33.1069,Y 128.7395,Z 176,A 76.7638,B 7.2168,C 0.0854,E1 7.2572,E2 375.1174} C_DIS
LIN {X 29.1307,Y 129.6973,Z 176,A 78.5129,B 7.2168,C 0.0845,E1 7.2525,E2 373.3705} C_DIS
LIN {X 25.2387,Y 130.51,Z 176,A 80.138,B 7.2168,C 0.0849,E1 7.248,E2 371.7564} C_DIS
LIN {X 21.8887,Y 131.1132,Z 176,A 81.5615,B 7.2168,C 0.0849,E1 7.2441,E2 370.3385} C_DIS
LIN {X 18.5958,Y 131.6208,Z 176,A 82.976,B 7.2168,C 0.0846,E1 7.2402,E2 368.9271} C_DIS
LIN {X 14.6605,Y 132.1177,Z 176,A 84.6961,B 7.2168,C 0.0838,E1 7.2355,E2 367.2064} C_DIS
LIN {X 10.7008,Y 132.4974,Z 176,A 86.4158,B 7.2168,C 0.0833,E1 7.2307,E2 365.4867} C_DIS
LIN {X 7.2333,Y 132.7322,Z 176,A 87.837,B 7.2168,C 0.0842,E1 7.2267,E2 364.0752} C_DIS
LIN {X 3.9794,Y 132.8687,Z 176,A 89.3041,B 7.2168,C 0.0831,E1 7.2226,E2 362.6011} C_DIS
LIN {X 0.0184,Y 132.93,Z 176,A 91.0239,B 7.2168,C 0.0828,E1 7.2178,E2 360.8807} C_DIS
LIN {X -3.2621,Y 132.8886,Z 176,A 92.4322,B 7.2168,C 0.083,E1 7.2139,E2 359.4737} C_DIS
LIN {X -6.5184,Y 132.7681,Z 176,A 93.9253,B 7.2168,C 0.0818,E1 7.2097,E2 357.9707} C_DIS
LIN {X -10.6863,Y 132.4986,Z 176,A 95.6401,B 7.2168,C 0.0835,E1 7.205,E2 356.267} C_DIS
LIN {X -13.7245,Y 132.2184,Z 176,A 97.0113,B 7.2168,C 0.083,E1 7.2011,E2 354.8899} C_DIS
LIN {X -17.8882,Y 131.7201,Z 176,A 98.7452,B 7.2168,C 0.0847,E1 7.1964,E2 353.1657} C_DIS
LIN {X -21.1123,Y 131.2427,Z 176,A 100.152,B 7.2168,C 0.0853,E1 7.1925,E2 351.7594} C_DIS
LIN {X -25.2273,Y 130.5122,Z 176,A 101.9719,B 7.2168,C 0.086,E1 7.1875,E2 349.9384} C_DIS
LIN {X -29.1088,Y 129.7023,Z 176,A 103.7019,B 7.2168,C 0.0867,E1 7.1827,E2 348.207} C_DIS
LIN {X -32.9801,Y 128.7717,Z 176,A 105.4379,B 7.2168,C 0.0876,E1 7.178,E2 346.4697} C_DIS
LIN {X -36.3363,Y 127.866,Z 176,A 107.082,B 7.2168,C 0.0867,E1 7.1736,E2 344.8093} C_DIS
LIN {X -40.1508,Y 126.7192,Z 176,A 108.6799,B 7.2168,C 0.0898,E1 7.1693,E2 343.2267} C_DIS
LIN {X -44.1045,Y 125.3989,Z 176,A 110.4598,B 7.2168,C 0.0917,E1 7.1646,E2 341.45} C_DIS
LIN {X -46.9472,Y 124.3616,Z 176,A 111.7955,B 7.2168,C 0.0926,E1 7.1611,E2 340.1115} C_DIS
LIN {X -50.1623,Y 123.1004,Z 176,A 113.2747,B 7.2168,C 0.0943,E1 7.1573,E2 338.6345} C_DIS
LIN {X -53.1332,Y 121.8472,Z 176,A 114.8251,B 7.2168,C 0.0937,E1 7.1533,E2 337.0661} C_DIS
LIN {X -57.4641,Y 119.8649,Z 176,A 116.7466,B 7.2167,C 0.098,E1 7.1485,E2 335.1617} C_DIS
LIN {X -60.6006,Y 118.3104,Z 176,A 118.3608,B 7.2167,C 0.0985,E1 7.1444,E2 333.5362} C_DIS
LIN {X -64.0958,Y 116.4563,Z 176,A 120.128,B 7.2167,C 0.1,E1 7.1401,E2 331.763} C_DIS
LIN {X -67.7193,Y 114.3874,Z 176,A 121.8072,B 7.2166,C 0.1042,E1 7.136,E2 330.0995} C_DIS
LIN {X -70.4949,Y 112.6978,Z 176,A 123.2268,B 7.2166,C 0.1061,E1 7.1327,E2 328.6788} C_DIS
LIN {X -73.2264,Y 110.9421,Z 176,A 124.6477,B 7.2166,C 0.108,E1 7.1293,E2 327.2566} C_DIS
LIN {X -76.5494,Y 108.6758,Z 176,A 126.5222,B 7.2166,C 0.109,E1 7.125,E2 325.3667} C_DIS
LIN {X -79.9289,Y 106.215,Z 176,A 128.2669,B 7.2165,C 0.1128,E1 7.1211,E2 323.6304} C_DIS
LIN {X -83.0569,Y 103.7877,Z 176,A 130.0198,B 7.2165,C 0.1153,E1 7.1173,E2 321.8735} C_DIS
LIN {X -86.206,Y 101.1868,Z 176,A 131.8142,B 7.2164,C 0.1181,E1 7.1134,E2 320.0765} C_DIS
LIN {X -89.5339,Y 98.2547,Z 176,A 133.7605,B 7.2164,C 0.1213,E1 7.1094,E2 318.1279} C_DIS
LIN {X -92.5758,Y 95.3938,Z 176,A 135.5469,B 7.2163,C 0.1251,E1 7.1058,E2 316.3447} C_DIS
LIN {X -95.3874,Y 92.5824,Z 176,A 137.3217,B 7.2163,C 0.1278,E1 7.1023,E2 314.5643} C_DIS
LIN {X -98.2607,Y 89.5272,Z 176,A 139.1438,B 7.2161,C 0.1315,E1 7.0988,E2 312.742} C_DIS
LIN {X -100.8818,Y 86.563,Z 176,A 140.8907,B 7.2161,C 0.1347,E1 7.0956,E2 310.9918} C_DIS
LIN {X -103.4822,Y 83.4365,Z 176,A 142.6598,B 7.2161,C 0.1384,E1 7.0925,E2 309.2224} C_DIS
LIN {X -106.2192,Y 79.9234,Z 176,A 144.5684,B 7.2159,C 0.1429,E1 7.0892,E2 307.3169} C_DIS
LIN {X -108.2724,Y 77.1193,Z 176,A 146.1838,B 7.2159,C 0.1449,E1 7.0866,E2 305.689} C_DIS
LIN {X -110.926,Y 73.2508,Z 176,A 148.2253,B 7.2158,C 0.1495,E1 7.0834,E2 303.647} C_DIS
LIN {X -113.1558,Y 69.7572,Z 176,A 150.0605,B 7.2158,C 0.1533,E1 7.0807,E2 301.8077} C_DIS
LIN {X -115.2522,Y 66.2369,Z 176,A 151.8746,B 7.2156,C 0.1571,E1 7.0781,E2 299.9895} C_DIS
LIN {X -117.2265,Y 62.6758,Z 176,A 153.7014,B 7.2156,C 0.1607,E1 7.0757,E2 298.1558} C_DIS
LIN {X -119.1453,Y 58.9415,Z 176,A 155.3579,B 7.2154,C 0.1672,E1 7.0736,E2 296.5193} C_DIS
LIN {X -120.8501,Y 55.364,Z 176,A 157.1046,B 7.2154,C 0.1712,E1 7.0715,E2 294.7697} C_DIS
LIN {X -122.1703,Y 52.386,Z 176,A 158.5031,B 7.2152,C 0.175,E1 7.07,E2 293.3731} C_DIS
LIN {X -123.4235,Y 49.3608,Z 176,A 159.9723,B 7.2152,C 0.1781,E1 7.0684,E2 291.8984} C_DIS
LIN {X -124.6024,Y 46.3041,Z 176,A 161.5292,B 7.2151,C 0.1801,E1 7.0669,E2 290.3254} C_DIS
LIN {X -125.998,Y 42.3602,Z 176,A 163.3911,B 7.215,C 0.1843,E1 7.0652,E2 288.4583} C_DIS
LIN {X -127.2036,Y 38.5885,Z 176,A 164.9891,B 7.2148,C 0.1904,E1 7.0639,E2 286.8749} C_DIS
LIN {X -128.2966,Y 34.7856,Z 176,A 166.7957,B 7.2148,C 0.1939,E1 7.0625,E2 285.0577} C_DIS
LIN {X -129.1613,Y 31.4195,Z 176,A 168.2601,B 7.2146,C 0.1985,E1 7.0615,E2 283.5987} C_DIS
LIN {X -130.0411,Y 27.5559,Z 176,A 169.9973,B 7.2145,C 0.2029,E1 7.0605,E2 281.8596} C_DIS
LIN {X -130.6845,Y 24.3261,Z 176,A 171.4406,B 7.2144,C 0.2067,E1 7.0597,E2 280.4148} C_DIS
LIN {X -131.2424,Y 21.1145,Z 176,A 172.868,B 7.2143,C 0.2104,E1 7.0591,E2 278.9859} C_DIS
LIN {X -131.8403,Y 16.9714,Z 176,A 174.8562,B 7.2142,C 0.2133,E1 7.0583,E2 276.9772} C_DIS
LIN {X -132.2878,Y 13.0328,Z 176,A 176.5832,B 7.2141,C 0.218,E1 7.0578,E2 275.2494} C_DIS
LIN {X -132.6347,Y 8.8497,Z 176,A 178.3365,B 7.2139,C 0.2239,E1 7.0574,E2 273.5045} C_DIS
LIN {X -132.8022,Y 5.8143,Z 176,A 179.7326,B 7.2138,C 0.2266,E1 7.0572,E2 272.0992} C_DIS
LIN {X -132.9075,Y 2.3376,Z 176,A -178.7881,B 7.2136,C 0.2311,E1 7.0572,E2 270.6236} C_DIS
LIN {X -132.9193,Y -1.6264,Z 176,A -177.0512,B 7.2136,C 0.2357,E1 7.0572,E2 268.8847} C_DIS
LIN {X -132.838,Y -4.8965,Z 176,A -175.6228,B 7.2134,C 0.2395,E1 7.0572,E2 267.4552} C_DIS
LIN {X -132.6344,Y -8.8547,Z 176,A -173.8183,B 7.2133,C 0.2433,E1 7.0576,E2 265.6405} C_DIS
LIN {X -132.2885,Y -13.0255,Z 176,A -172.0535,B 7.2131,C 0.2489,E1 7.058,E2 263.8819} C_DIS
LIN {X -131.8991,Y -16.523,Z 176,A -170.3564,B 7.213,C 0.251,E1 7.0586,E2 262.1641} C_DIS
LIN {X -131.3837,Y -20.2026,Z 176,A -168.8503,B 7.2128,C 0.2567,E1 7.0592,E2 260.6707} C_DIS
LIN {X -130.8487,Y -23.4179,Z 176,A -167.393,B 7.2127,C 0.26,E1 7.0599,E2 259.2082} C_DIS
LIN {X -130.191,Y -26.8362,Z 176,A -165.8989,B 7.2125,C 0.2643,E1 7.0607,E2 257.7159} C_DIS
LIN {X -129.3384,Y -30.6848,Z 176,A -164.168,B 7.2124,C 0.2686,E1 7.0618,E2 255.9825} C_DIS
LIN {X -128.5641,Y -33.7823,Z 176,A -162.7801,B 7.2122,C 0.2723,E1 7.0628,E2 254.5941} C_DIS
LIN {X -127.6348,Y -37.1369,Z 176,A -161.0949,B 7.2122,C 0.2741,E1 7.0641,E2 252.8874} C_DIS
LIN {X -126.5061,Y -40.8179,Z 176,A -159.5375,B 7.2119,C 0.2799,E1 7.0654,E2 251.3436} C_DIS
LIN {X -125.3968,Y -44.1104,Z 176,A -157.8511,B 7.2119,C 0.2816,E1 7.0669,E2 249.6352} C_DIS
LIN {X -123.953,Y -48.0145,Z 176,A -156.1176,B 7.2116,C 0.2871,E1 7.0686,E2 247.9101} C_DIS
LIN {X -122.4522,Y -51.7249,Z 176,A -154.4201,B 7.2115,C 0.292,E1 7.0704,E2 246.2171} C_DIS
LIN {X -120.8556,Y -55.3522,Z 176,A -152.6343,B 7.2113,C 0.2955,E1 7.0725,E2 244.4228} C_DIS
LIN {X -119.145,Y -58.9422,Z 176,A -150.9042,B 7.2111,C 0.2996,E1 7.0746,E2 242.6916} C_DIS
LIN {X -117.5686,Y -62.0272,Z 176,A -149.4848,B 7.2109,C 0.3043,E1 7.0764,E2 241.2821} C_DIS
LIN {X -115.6794,Y -65.488,Z 176,A -147.6831,B 7.2109,C 0.3072,E1 7.0789,E2 239.4688} C_DIS
LIN {X -113.9027,Y -68.5309,Z 176,A -146.0067,B 7.2108,C 0.3089,E1 7.0813,E2 237.7738} C_DIS
LIN {X -111.8099,Y -71.8948,Z 176,A -144.4013,B 7.2105,C 0.3143,E1 7.0837,E2 236.1818} C_DIS
LIN {X -110.0142,Y -74.6131,Z 176,A -142.8362,B 7.2105,C 0.3155,E1 7.0861,E2 234.5976} C_DIS
LIN {X -107.3223,Y -78.4363,Z 176,A -140.8243,B 7.2103,C 0.3201,E1 7.0894,E2 232.587} C_DIS
LIN {X -105.0883,Y -81.4044,Z 176,A -139.2222,B 7.2101,C 0.3236,E1 7.0921,E2 230.9854} C_DIS
LIN {X -102.5525,Y -84.577,Z 176,A -137.4218,B 7.21,C 0.3268,E1 7.0953,E2 229.1795} C_DIS
LIN {X -99.8183,Y -87.7875,Z 176,A -135.5956,B 7.2098,C 0.3305,E1 7.0986,E2 227.3529} C_DIS
LIN {X -97.0732,Y -90.8137,Z 176,A -133.7895,B 7.2097,C 0.3335,E1 7.1021,E2 225.5418} C_DIS
LIN {X -93.9986,Y -93.9929,Z 176,A -131.8738,B 7.2095,C 0.3372,E1 7.1058,E2 223.6255} C_DIS
LIN {X -91.0756,Y -96.8271,Z 176,A -130.093,B 7.2094,C 0.3402,E1 7.1094,E2 221.8419} C_DIS
LIN {X -88.0552,Y -99.5816,Z 176,A -128.3301,B 7.2092,C 0.3434,E1 7.1131,E2 220.0792} C_DIS
LIN {X -84.9622,Y -102.2336,Z 176,A -126.5401,B 7.2091,C 0.346,E1 7.1169,E2 218.2855} C_DIS
LIN {X -81.7787,Y -104.7981,Z 176,A -124.6831,B 7.209,C 0.3477,E1 7.121,E2 216.417} C_DIS
LIN {X -78.4561,Y -107.3077,Z 176,A -123.0109,B 7.2088,C 0.3523,E1 7.1247,E2 214.7601} C_DIS
LIN {X -75.7829,Y -109.2118,Z 176,A -121.445,B 7.2088,C 0.3525,E1 7.1283,E2 213.1757} C_DIS
LIN {X -72.6035,Y -111.3509,Z 176,A -119.8859,B 7.2086,C 0.3562,E1 7.132,E2 211.6282} C_DIS
LIN {X -69.7386,Y -113.1673,Z 176,A -118.3066,B 7.2086,C 0.3567,E1 7.1357,E2 210.0345} C_DIS
LIN {X -66.1491,Y -115.3024,Z 176,A -116.6244,B 7.2084,C 0.3608,E1 7.1398,E2 208.3669} C_DIS
LIN {X -62.6571,Y -117.2366,Z 176,A -114.7025,B 7.2084,C 0.3601,E1 7.1445,E2 206.4201} C_DIS
LIN {X -58.9364,Y -119.1478,Z 176,A -113.067,B 7.2082,C 0.3646,E1 7.1486,E2 204.8051} C_DIS
LIN {X -55.3575,Y -120.8531,Z 176,A -111.2103,B 7.2082,C 0.3644,E1 7.1533,E2 202.93} C_DIS
LIN {X -51.2942,Y -122.6321,Z 176,A -109.3394,B 7.208,C 0.367,E1 7.1581,E2 201.0641} C_DIS
LIN {X -47.8445,Y -124.0191,Z 176,A -107.8021,B 7.208,C 0.3694,E1 7.1621,E2 199.5347} C_DIS
LIN {X -44.6967,Y -125.1883,Z 176,A -106.1897,B 7.208,C 0.3683,E1 7.1664,E2 197.9015} C_DIS
LIN {X -40.1743,Y -126.7117,Z 176,A -104.2803,B 7.2078,C 0.372,E1 7.1714,E2 196.0101} C_DIS
LIN {X -37.0844,Y -127.6502,Z 176,A -102.8837,B 7.2078,C 0.373,E1 7.1751,E2 194.6126} C_DIS
LIN {X -34.0111,Y -128.5031,Z 176,A -101.4458,B 7.2078,C 0.3729,E1 7.179,E2 193.1665} C_DIS
LIN {X -29.8156,Y -129.5409,Z 176,A -99.6242,B 7.2077,C 0.3745,E1 7.184,E2 191.3496} C_DIS
LIN {X -25.9329,Y -130.3748,Z 176,A -97.9184,B 7.2077,C 0.3754,E1 7.1886,E2 189.6441} C_DIS
LIN {X -22.7309,Y -130.9716,Z 176,A -96.5142,B 7.2076,C 0.376,E1 7.1925,E2 188.2395} C_DIS
LIN {X -19.5133,Y -131.4897,Z 176,A -95.0817,B 7.2076,C 0.376,E1 7.1964,E2 186.803} C_DIS
LIN {X -15.5874,Y -132.0108,Z 176,A -93.3612,B 7.2076,C 0.3762,E1 7.2012,E2 185.0801} C_DIS
LIN {X -11.4063,Y -132.4378,Z 176,A -91.4687,B 7.2076,C 0.3752,E1 7.2065,E2 183.1769} C_DIS
LIN {X -7.2399,Y -132.7318,Z 176,A -89.8281,B 7.2075,C 0.3778,E1 7.211,E2 181.5555} C_DIS
LIN {X -3.9874,Y -132.8685,Z 176,A -88.3601,B 7.2075,C 0.3768,E1 7.2152,E2 180.0787} C_DIS
LIN {X -0.1907,Y -132.929,Z 176,A -86.6977,B 7.2075,C 0.3762,E1 7.2198,E2 178.4124} C_DIS
LIN {X -0.1907,Y -132.929,Z 176,A -86.6977,B 7.2075,C 0.3762,E1 7.2198,E2 178.4124} C_DIS
Enddeposition()
LIN {X 0.9741,Y -133.8293,Z 176,A -86.2359,B 7.2073,C 0.3809,E1 7.221,E2 177.9882} C_DIS
Startdeposition()
$VEL.CP = VEL_PRINT
LIN {X -2.0661,Y -133.8178,Z 176,A -88.2509,B 7.2067,C 0.3923,E1 7.2151,E2 180.0929} C_DIS
LIN {X -6.8438,Y -133.6586,Z 176,A -90.1799,B 7.2068,C 0.3905,E1 7.2098,E2 182.0083} C_DIS
LIN {X -10.4874,Y -133.4241,Z 176,A -91.8377,B 7.2068,C 0.3918,E1 7.2051,E2 183.6785} C_DIS
LIN {X -14.1916,Y -133.079,Z 176,A -93.4938,B 7.2068,C 0.3925,E1 7.2005,E2 185.343} C_DIS
LIN {X -18.65,Y -132.528,Z 176,A -95.2359,B 7.2069,C 0.3892,E1 7.1958,E2 187.0634} C_DIS
LIN {X -21.4931,Y -132.0974,Z 176,A -96.5737,B 7.2069,C 0.3905,E1 7.192,E2 188.4148} C_DIS
LIN {X -25.4688,Y -131.3881,Z 176,A -98.2853,B 7.2069,C 0.3895,E1 7.1873,E2 190.1248} C_DIS
LIN {X -29.5554,Y -130.5294,Z 176,A -100.0562,B 7.2069,C 0.3884,E1 7.1825,E2 191.8941} C_DIS
LIN {X -32.8324,Y -129.7436,Z 176,A -101.5024,B 7.2069,C 0.3876,E1 7.1786,E2 193.3411} C_DIS
LIN {X -35.7076,Y -128.9823,Z 176,A -103.1084,B 7.2068,C 0.3917,E1 7.1741,E2 194.9885} C_DIS
LIN {X -39.0535,Y -128.0085,Z 176,A -105.1169,B 7.2064,C 0.3981,E1 7.1686,E2 197.0606} C_DIS
LIN {X -44.9419,Y -126.0626,Z 176,A -107.1599,B 7.207,C 0.387,E1 7.1634,E2 199.0291} C_DIS
LIN {X -49.564,Y -124.3181,Z 176,A -109.0835,B 7.2073,C 0.3823,E1 7.1585,E2 200.9293} C_DIS
LIN {X -53.3559,Y -122.7376,Z 176,A -110.8667,B 7.2073,C 0.3809,E1 7.1539,E2 202.7156} C_DIS
LIN {X -57.2284,Y -120.9813,Z 176,A -112.625,B 7.2075,C 0.378,E1 7.1494,E2 204.4664} C_DIS
LIN {X -59.9681,Y -119.6488,Z 176,A -114.1179,B 7.2075,C 0.3791,E1 7.1456,E2 205.9828} C_DIS
LIN {X -63.7155,Y -117.696,Z 176,A -115.9438,B 7.2075,C 0.3771,E1 7.1411,E2 207.8107} C_DIS
LIN {X -67.4538,Y -115.594,Z 176,A -117.7962,B 7.2077,C 0.3749,E1 7.1366,E2 209.6651} C_DIS
LIN {X -71.3096,Y -113.2555,Z 176,A -119.7214,B 7.2078,C 0.3721,E1 7.1321,E2 211.5896} C_DIS
LIN {X -75.0012,Y -110.8452,Z 176,A -121.4854,B 7.208,C 0.3675,E1 7.128,E2 213.3383} C_DIS
LIN {X -79.6723,Y -107.5373,Z 176,A -124.1259,B 7.2081,C 0.3663,E1 7.122,E2 216.0018} C_DIS
LIN {X -82.399,Y -105.4626,Z 176,A -125.6998,B 7.2081,C 0.3653,E1 7.1185,E2 217.5887} C_DIS
LIN {X -86.1981,Y -102.3805,Z 176,A -127.6914,B 7.2084,C 0.3602,E1 7.1142,E2 219.5673} C_DIS
LIN {X -89.5786,Y -99.4367,Z 176,A -129.6154,B 7.2086,C 0.3568,E1 7.1102,E2 221.4915} C_DIS
LIN {X -92.6859,Y -96.5466,Z 176,A -131.4236,B 7.2088,C 0.3532,E1 7.1065,E2 223.2982} C_DIS
LIN {X -95.626,Y -93.635,Z 176,A -133.2215,B 7.2089,C 0.3501,E1 7.103,E2 225.0989} C_DIS
LIN {X -98.3633,Y -90.7555,Z 176,A -134.8199,B 7.2091,C 0.3453,E1 7.0999,E2 226.6842} C_DIS
LIN {X -100.6849,Y -88.1728,Z 176,A -136.538,B 7.2091,C 0.3453,E1 7.0967,E2 228.4301} C_DIS
LIN {X -103.6891,Y -84.6192,Z 176,A -138.6617,B 7.2093,C 0.3427,E1 7.0929,E2 230.5692} C_DIS
LIN {X -106.774,Y -80.6917,Z 176,A -140.5174,B 7.2096,C 0.3343,E1 7.0898,E2 232.3896} C_DIS
LIN {X -108.6077,Y -78.2073,Z 176,A -142.0481,B 7.2096,C 0.334,E1 7.0872,E2 233.9453} C_DIS
LIN {X -111.3018,Y -74.322,Z 176,A -144.0884,B 7.2099,C 0.3295,E1 7.084,E2 235.9867} C_DIS
LIN {X -113.5142,Y -70.8972,Z 176,A -145.8934,B 7.21,C 0.3261,E1 7.0813,E2 237.7981} C_DIS
LIN {X -115.1475,Y -68.213,Z 176,A -148.035,B 7.2097,C 0.3328,E1 7.0781,E2 240.0355} C_DIS
LIN {X -118.168,Y -62.8338,Z 176,A -149.9318,B 7.2104,C 0.317,E1 7.0757,E2 241.8409} C_DIS
LIN {X -119.7675,Y -59.7276,Z 176,A -151.6699,B 7.2104,C 0.3162,E1 7.0735,E2 243.6077} C_DIS
LIN {X -121.1931,Y -56.7801,Z 176,A -152.7992,B 7.2108,C 0.3092,E1 7.0722,E2 244.7032} C_DIS
LIN {X -122.6805,Y -53.4881,Z 176,A -154.4387,B 7.2108,C 0.3064,E1 7.0703,E2 246.353} C_DIS
LIN {X -123.99,Y -50.3779,Z 176,A -155.8874,B 7.211,C 0.3026,E1 7.0688,E2 247.8012} C_DIS
LIN {X -125.1481,Y -47.4294,Z 176,A -157.254,B 7.2112,C 0.2992,E1 7.0674,E2 249.1684} C_DIS
LIN {X -126.3535,Y -44.1158,Z 176,A -158.5766,B 7.2114,C 0.2928,E1 7.0662,E2 250.4673} C_DIS
LIN {X -127.3335,Y -41.2041,Z 176,A -160.1272,B 7.2114,C 0.2922,E1 7.0648,E2 252.0456} C_DIS
LIN {X -128.5932,Y -37.0867,Z 176,A -162.1896,B 7.2116,C 0.2898,E1 7.0631,E2 254.1332} C_DIS
LIN {X -130.126,Y -31.2826,Z 176,A -164.771,B 7.2118,C 0.2828,E1 7.0614,E2 256.7142} C_DIS
LIN {X -131.2859,Y -25.9977,Z 176,A -167.0528,B 7.2121,C 0.2759,E1 7.06,E2 258.9902} C_DIS
LIN {X -131.9778,Y -22.2098,Z 176,A -168.6824,B 7.2123,C 0.2711,E1 7.0593,E2 260.6162} C_DIS
LIN {X -132.5817,Y -18.2737,Z 176,A -170.5213,B 7.2124,C 0.2679,E1 7.0585,E2 262.47} C_DIS
LIN {X -133.0596,Y -14.3719,Z 176,A -172.1133,B 7.2126,C 0.262,E1 7.058,E2 264.0496} C_DIS
LIN {X -133.4137,Y -10.6129,Z 176,A -173.8917,B 7.2127,C 0.2593,E1 7.0576,E2 265.8464} C_DIS
LIN {X -133.6844,Y -6.33,Z 176,A -175.7448,B 7.2129,C 0.2542,E1 7.0573,E2 267.6999} C_DIS
LIN {X -133.8125,Y -2.389,Z 176,A -177.4054,B 7.2131,C 0.2491,E1 7.0572,E2 269.3557} C_DIS
LIN {X -133.8188,Y 2.0113,Z 176,A -179.3184,B 7.2133,C 0.244,E1 7.0572,E2 271.2707} C_DIS
LIN {X -133.696,Y 6.099,Z 176,A 178.8242,B 7.2133,C 0.2402,E1 7.0574,E2 273.1394} C_DIS
LIN {X -133.4689,Y 9.874,Z 176,A 177.2389,B 7.2135,C 0.2352,E1 7.0577,E2 274.7191} C_DIS
LIN {X -133.0944,Y 14.0486,Z 176,A 175.4128,B 7.2137,C 0.2304,E1 7.0582,E2 276.5475} C_DIS
LIN {X -132.6137,Y 18.0403,Z 176,A 173.6234,B 7.2138,C 0.2263,E1 7.0588,E2 278.3436} C_DIS
LIN {X -131.9833,Y 22.177,Z 176,A 171.8711,B 7.214,C 0.2208,E1 7.0596,E2 280.0895} C_DIS
LIN {X -131.3011,Y 25.9233,Z 176,A 170.0628,B 7.214,C 0.2183,E1 7.0605,E2 281.9177} C_DIS
LIN {X -130.4907,Y 29.7244,Z 176,A 168.3959,B 7.2142,C 0.2136,E1 7.0615,E2 283.5833} C_DIS
LIN {X -129.4869,Y 33.837,Z 176,A 166.5919,B 7.2144,C 0.2085,E1 7.0628,E2 285.3848} C_DIS
LIN {X -128.491,Y 37.4359,Z 176,A 165.0006,B 7.2144,C 0.204,E1 7.064,E2 286.9736} C_DIS
LIN {X -127.6249,Y 40.2917,Z 176,A 163.6898,B 7.2146,C 0.2008,E1 7.0651,E2 288.2873} C_DIS
LIN {X -126.4742,Y 43.7678,Z 176,A 162.1124,B 7.2146,C 0.1967,E1 7.0665,E2 289.8643} C_DIS
LIN {X -125.0179,Y 47.7748,Z 176,A 160.2144,B 7.2148,C 0.1926,E1 7.0683,E2 291.7693} C_DIS
LIN {X -123.5665,Y 51.4068,Z 176,A 158.5125,B 7.2149,C 0.1885,E1 7.0701,E2 293.4728} C_DIS
LIN {X -122.2751,Y 54.4075,Z 176,A 157.111,B 7.215,C 0.1848,E1 7.0717,E2 294.8733} C_DIS
LIN {X -120.8067,Y 57.5939,Z 176,A 155.5358,B 7.215,C 0.1818,E1 7.0736,E2 296.4558} C_DIS
LIN {X -119.0387,Y 61.1665,Z 176,A 153.8411,B 7.2152,C 0.1772,E1 7.0757,E2 298.1475} C_DIS
LIN {X -117.1378,Y 64.7346,Z 176,A 151.7497,B 7.2152,C 0.1772,E1 7.0785,E2 300.2801} C_DIS
LIN {X -115.4385,Y 67.7185,Z 176,A 149.9036,B 7.2152,C 0.1782,E1 7.0812,E2 302.1691} C_DIS
LIN {X -112.7096,Y 72.1691,Z 176,A 148.482,B 7.2155,C 0.1627,E1 7.0832,E2 303.4924} C_DIS
LIN {X -109.6439,Y 76.7477,Z 176,A 145.8408,B 7.2155,C 0.1606,E1 7.0874,E2 306.165} C_DIS
LIN {X -107.2638,Y 80.0396,Z 176,A 144.1242,B 7.2157,C 0.1563,E1 7.0902,E2 307.8773} C_DIS
LIN {X -104.7456,Y 83.3078,Z 176,A 142.4494,B 7.2157,C 0.1511,E1 7.0931,E2 309.5396} C_DIS
LIN {X -102.4036,Y 86.1706,Z 176,A 140.6473,B 7.2157,C 0.1503,E1 7.0963,E2 311.3662} C_DIS
LIN {X -99.5007,Y 89.5071,Z 176,A 138.8633,B 7.2159,C 0.1449,E1 7.0996,E2 313.1354} C_DIS
LIN {X -96.925,Y 92.2899,Z 176,A 137.0526,B 7.2159,C 0.1438,E1 7.1031,E2 314.9668} C_DIS
LIN {X -93.532,Y 95.7271,Z 176,A 135.017,B 7.216,C 0.1392,E1 7.1071,E2 316.9968} C_DIS
LIN {X -90.4705,Y 98.6252,Z 176,A 133.225,B 7.216,C 0.1355,E1 7.1107,E2 318.7856} C_DIS
LIN {X -87.4624,Y 101.3024,Z 176,A 131.3992,B 7.2161,C 0.1335,E1 7.1146,E2 320.6219} C_DIS
LIN {X -84.0921,Y 104.1171,Z 176,A 129.5219,B 7.2161,C 0.13,E1 7.1186,E2 322.4973} C_DIS
LIN {X -81.0012,Y 106.5401,Z 176,A 127.8371,B 7.2162,C 0.1271,E1 7.1224,E2 324.1811} C_DIS
LIN {X -78.0471,Y 108.7224,Z 176,A 126.3596,B 7.2163,C 0.1232,E1 7.1257,E2 325.646} C_DIS
LIN {X -74.885,Y 110.9239,Z 176,A 124.5208,B 7.2163,C 0.123,E1 7.1299,E2 327.5058} C_DIS
LIN {X -70.321,Y 113.8725,Z 176,A 122.2193,B 7.2163,C 0.1191,E1 7.1354,E2 329.8025} C_DIS
LIN {X -66.8756,Y 115.929,Z 176,A 120.5389,B 7.2164,C 0.1161,E1 7.1394,E2 331.4771} C_DIS
LIN {X -64.0137,Y 117.5334,Z 176,A 119.0636,B 7.2164,C 0.1151,E1 7.143,E2 332.9595} C_DIS
LIN {X -61.535,Y 118.85,Z 176,A 117.6049,B 7.2164,C 0.1169,E1 7.1467,E2 334.4477} C_DIS
LIN {X -56.6255,Y 121.2646,Z 176,A 115.6491,B 7.2165,C 0.1088,E1 7.1515,E2 336.3561} C_DIS
LIN {X -53.3959,Y 122.7203,Z 176,A 114.2235,B 7.2165,C 0.1058,E1 7.1551,E2 337.7698} C_DIS
LIN {X -48.431,Y 124.7628,Z 176,A 111.4721,B 7.2165,C 0.1095,E1 7.1624,E2 340.573} C_DIS
LIN {X -43.9479,Y 126.4117,Z 176,A 109.7378,B 7.2166,C 0.1032,E1 7.1668,E2 342.2692} C_DIS
LIN {X -41.1097,Y 127.3636,Z 176,A 108.5211,B 7.2166,C 0.1012,E1 7.17,E2 343.4773} C_DIS
LIN {X -36.4636,Y 128.7709,Z 176,A 106.1801,B 7.2166,C 0.1032,E1 7.1764,E2 345.8481} C_DIS
LIN {X -32.9186,Y 129.7217,Z 176,A 104.6905,B 7.2166,C 0.1009,E1 7.1804,E2 347.327} C_DIS
LIN {X -29.2612,Y 130.5966,Z 176,A 102.9747,B 7.2166,C 0.1013,E1 7.1851,E2 349.0544} C_DIS
LIN {X -25.3539,Y 131.4101,Z 176,A 101.3888,B 7.2166,C 0.0986,E1 7.1894,E2 350.6247} C_DIS
LIN {X -21.8654,Y 132.0353,Z 176,A 99.8008,B 7.2166,C 0.0989,E1 7.1938,E2 352.2201} C_DIS
LIN {X -17.8083,Y 132.6441,Z 176,A 98.0457,B 7.2166,C 0.0982,E1 7.1986,E2 353.9741} C_DIS
LIN {X -14.5683,Y 133.0385,Z 176,A 96.5745,B 7.2166,C 0.0988,E1 7.2027,E2 355.4533} C_DIS
LIN {X -10.412,Y 133.4296,Z 176,A 94.7854,B 7.2166,C 0.0984,E1 7.2077,E2 357.2417} C_DIS
LIN {X -6.4621,Y 133.6778,Z 176,A 93.1728,B 7.2167,C 0.0969,E1 7.2122,E2 358.8439} C_DIS
LIN {X -2.6462,Y 133.8082,Z 176,A 91.6038,B 7.2167,C 0.0958,E1 7.2165,E2 360.4043} C_DIS
LIN {X 1.0284,Y 133.8301,Z 176,A 89.8598,B 7.2167,C 0.0984,E1 7.2214,E2 362.1677} C_DIS
LIN {X 5.3307,Y 133.7275,Z 176,A 88.1031,B 7.2167,C 0.0973,E1 7.2263,E2 363.9136} C_DIS
LIN {X 9.2176,Y 133.5168,Z 176,A 86.4014,B 7.2167,C 0.0981,E1 7.2311,E2 365.6188} C_DIS
LIN {X 14.325,Y 133.0647,Z 176,A 84.2649,B 7.2167,C 0.0978,E1 7.237,E2 367.7475} C_DIS
LIN {X 18.2337,Y 132.5875,Z 176,A 82.4697,B 7.2167,C 0.1001,E1 7.242,E2 369.5551} C_DIS
LIN {X 22.4484,Y 131.938,Z 176,A 80.7307,B 7.2167,C 0.0996,E1 7.2468,E2 371.2833} C_DIS
LIN {X 26.4302,Y 131.1979,Z 176,A 79.0286,B 7.2167,C 0.1001,E1 7.2514,E2 372.9811} C_DIS
LIN {X 29.5832,Y 130.523,Z 176,A 77.6892,B 7.2167,C 0.1003,E1 7.2551,E2 374.3153} C_DIS
LIN {X 32.5357,Y 129.8189,Z 176,A 76.0203,B 7.2166,C 0.107,E1 7.2597,E2 376.0275} C_DIS
LIN {X 35.9323,Y 128.9195,Z 176,A 74.0034,B 7.2164,C 0.1162,E1 7.2653,E2 378.1042} C_DIS
LIN {X 41.9663,Y 127.0837,Z 176,A 71.9657,B 7.2165,C 0.1082,E1 7.2705,E2 380.0637} C_DIS
LIN {X 46.5719,Y 125.4693,Z 176,A 70.1035,B 7.2165,C 0.1066,E1 7.2753,E2 381.8987} C_DIS
LIN {X 50.5913,Y 123.904,Z 176,A 68.2012,B 7.2165,C 0.1094,E1 7.2803,E2 383.8075} C_DIS
LIN {X 54.2823,Y 122.3311,Z 176,A 66.5088,B 7.2165,C 0.111,E1 7.2846,E2 385.4967} C_DIS
LIN {X 57.3544,Y 120.9211,Z 176,A 65.1622,B 7.2165,C 0.1111,E1 7.288,E2 386.8313} C_DIS
LIN {X 60.5425,Y 119.3564,Z 176,A 63.6446,B 7.2165,C 0.113,E1 7.2918,E2 388.3485} C_DIS
LIN {X 63.7531,Y 117.6755,Z 176,A 61.9668,B 7.2165,C 0.1172,E1 7.2959,E2 390.0415} C_DIS
LIN {X 67.6789,Y 115.4618,Z 176,A 60.1543,B 7.2164,C 0.118,E1 7.3003,E2 391.8401} C_DIS
LIN {X 71.2481,Y 113.2943,Z 176,A 58.3062,B 7.2164,C 0.1217,E1 7.3047,E2 393.6954} C_DIS
LIN {X 77.9063,Y 108.823,Z 176,A 54.9836,B 7.2163,C 0.1254,E1 7.3123,E2 397.0052} C_DIS
LIN {X 81.7938,Y 105.9324,Z 176,A 52.8853,B 7.2163,C 0.1294,E1 7.317,E2 399.1067} C_DIS
LIN {X 85.2057,Y 103.2078,Z 176,A 51.0258,B 7.2161,C 0.1326,E1 7.321,E2 400.9654} C_DIS
LIN {X 88.2348,Y 100.6308,Z 176,A 49.3338,B 7.2161,C 0.1356,E1 7.3246,E2 402.6565} C_DIS
LIN {X 91.465,Y 97.7042,Z 176,A 47.4886,B 7.2161,C 0.1389,E1 7.3284,E2 404.4996} C_DIS
LIN {X 94.7066,Y 94.5654,Z 176,A 45.6381,B 7.216,C 0.1413,E1 7.3321,E2 406.341} C_DIS
LIN {X 97.8683,Y 91.2887,Z 176,A 43.6811,B 7.2159,C 0.1455,E1 7.3358,E2 408.2994} C_DIS
LIN {X 101.0122,Y 87.7977,Z 176,A 41.8592,B 7.2159,C 0.1465,E1 7.3392,E2 410.0993} C_DIS
LIN {X 106.7067,Y 80.781,Z 176,A 38.0134,B 7.2157,C 0.1548,E1 7.3459,E2 413.9439} C_DIS
LIN {X 109.2151,Y 77.3561,Z 176,A 36.1066,B 7.2156,C 0.1606,E1 7.349,E2 415.8623} C_DIS
LIN {X 111.7024,Y 73.7186,Z 176,A 34.3351,B 7.2156,C 0.163,E1 7.3518,E2 417.6207} C_DIS
LIN {X 113.7918,Y 70.4511,Z 176,A 32.6636,B 7.2154,C 0.1672,E1 7.3543,E2 419.2944} C_DIS
LIN {X 115.8029,Y 67.0934,Z 176,A 30.9932,B 7.2154,C 0.1713,E1 7.3566,E2 420.965} C_DIS
LIN {X 117.9627,Y 63.2191,Z 176,A 29.0891,B 7.2152,C 0.1761,E1 7.3592,E2 422.8706} C_DIS
LIN {X 119.8786,Y 59.5023,Z 176,A 27.4607,B 7.2152,C 0.1778,E1 7.3612,E2 424.4805} C_DIS
LIN {X 121.3629,Y 56.4128,Z 176,A 25.9375,B 7.2151,C 0.1826,E1 7.363,E2 426.0112} C_DIS
LIN {X 122.9058,Y 52.9669,Z 176,A 24.432,B 7.215,C 0.1848,E1 7.3647,E2 427.5042} C_DIS
LIN {X 124.2837,Y 49.6493,Z 176,A 22.0994,B 7.2145,C 0.2032,E1 7.3673,E2 429.9333} C_DIS
LIN {X 126.3916,Y 44.0058,Z 176,A 20.4905,B 7.2148,C 0.1927,E1 7.3687,E2 431.4272} C_DIS
LIN {X 127.8838,Y 39.4609,Z 176,A 18.3618,B 7.2146,C 0.1997,E1 7.3705,E2 433.5671} C_DIS
LIN {X 128.7212,Y 36.6412,Z 176,A 17.171,B 7.2146,C 0.2019,E1 7.3714,E2 434.7505} C_DIS
LIN {X 129.6024,Y 33.3889,Z 176,A 15.6922,B 7.2144,C 0.2066,E1 7.3725,E2 436.2347} C_DIS
LIN {X 130.4566,Y 29.874,Z 176,A 14.2456,B 7.2144,C 0.209,E1 7.3734,E2 437.67} C_DIS
LIN {X 131.171,Y 26.5626,Z 176,A 12.806,B 7.2142,C 0.2129,E1 7.3742,E2 439.1094} C_DIS
LIN {X 131.8563,Y 22.9287,Z 176,A 11.0873,B 7.214,C 0.2199,E1 7.3751,E2 440.8458} C_DIS
LIN {X 132.4762,Y 19.0121,Z 176,A 9.6381,B 7.214,C 0.2201,E1 7.3757,E2 442.266} C_DIS
LIN {X 132.8892,Y 15.8703,Z 176,A 8.1945,B 7.2138,C 0.2256,E1 7.3762,E2 443.7213} C_DIS
LIN {X 133.2975,Y 11.9891,Z 176,A 6.4899,B 7.2137,C 0.231,E1 7.3766,E2 445.4314} C_DIS
LIN {X 133.5971,Y 7.9574,Z 176,A 4.9077,B 7.2137,C 0.2332,E1 7.3769,E2 446.9969} C_DIS
LIN {X 133.7718,Y 4.0852,Z 176,A 3.2148,B 7.2134,C 0.2386,E1 7.3771,E2 448.6952} C_DIS
LIN {X 133.8319,Y 0.8418,Z 176,A 1.9215,B 7.2134,C 0.2408,E1 7.3771,E2 449.978} C_DIS
LIN {X 133.8014,Y -3.0224,Z 176,A 0.1922,B 7.2131,C 0.247,E1 7.3771,E2 451.7179} C_DIS
LIN {X 133.6941,Y -6.1371,Z 176,A -1.2752,B 7.2129,C 0.2533,E1 7.3769,E2 453.2027} C_DIS
LIN {X 133.361,Y -11.2366,Z 176,A -3.1985,B 7.2129,C 0.2547,E1 7.3765,E2 455.0956} C_DIS
LIN {X 132.9713,Y -15.1826,Z 176,A -4.8929,B 7.2127,C 0.2595,E1 7.376,E2 456.7911} C_DIS
LIN {X 132.565,Y -18.3909,Z 176,A -6.2389,B 7.2126,C 0.2627,E1 7.3755,E2 458.1337} C_DIS
LIN {X 132.0188,Y -21.964,Z 176,A -7.6945,B 7.2125,C 0.2655,E1 7.3749,E2 459.5795} C_DIS
LIN {X 131.4692,Y -25.0445,Z 176,A -8.9555,B 7.2125,C 0.2678,E1 7.3742,E2 460.832} C_DIS
LIN {X 130.8617,Y -28.0468,Z 176,A -10.1422,B 7.2124,C 0.2692,E1 7.3736,E2 462.0046} C_DIS
LIN {X 129.768,Y -32.7362,Z 176,A -12.9103,B 7.2116,C 0.288,E1 7.3717,E2 464.8611} C_DIS
LIN {X 128.489,Y -37.4426,Z 176,A -14.5145,B 7.2118,C 0.285,E1 7.3705,E2 466.4081} C_DIS
LIN {X 127.3716,Y -41.0848,Z 176,A -16.0911,B 7.2116,C 0.2885,E1 7.3692,E2 467.9797} C_DIS
LIN {X 126.0193,Y -45.0621,Z 176,A -17.6197,B 7.2116,C 0.2885,E1 7.3678,E2 469.4768} C_DIS
LIN {X 124.8725,Y -48.1488,Z 176,A -19.1714,B 7.2114,C 0.2949,E1 7.3663,E2 471.0473} C_DIS
LIN {X 123.2354,Y -52.1997,Z 176,A -21.4068,B 7.2109,C 0.3066,E1 7.3638,E2 473.3293} C_DIS
LIN {X 121.5904,Y -55.921,Z 176,A -22.589,B 7.2111,C 0.301,E1 7.3625,E2 474.4445} C_DIS
LIN {X 119.1416,Y -60.9643,Z 176,A -25.0456,B 7.2108,C 0.3083,E1 7.3595,E2 476.9103} C_DIS
LIN {X 116.1603,Y -66.4729,Z 176,A -27.6945,B 7.2105,C 0.3146,E1 7.3559,E2 479.5579} C_DIS
LIN {X 114.2049,Y -69.7791,Z 176,A -29.1859,B 7.2105,C 0.3159,E1 7.3538,E2 481.032} C_DIS
LIN {X 112.419,Y -72.6215,Z 176,A -30.7365,B 7.2102,C 0.3216,E1 7.3514,E2 482.598} C_DIS
LIN {X 109.1102,Y -77.5046,Z 176,A -33.283,B 7.2099,C 0.3281,E1 7.3474,E2 485.1496} C_DIS
LIN {X 106.0457,Y -81.6475,Z 176,A -35.4584,B 7.2097,C 0.3327,E1 7.3437,E2 487.3233} C_DIS
LIN {X 103.259,Y -85.144,Z 176,A -37.3257,B 7.2096,C 0.3363,E1 7.3405,E2 489.1867} C_DIS
LIN {X 100.3882,Y -88.5103,Z 176,A -39.1714,B 7.2094,C 0.3396,E1 7.3371,E2 491.0282} C_DIS
LIN {X 97.4059,Y -91.7819,Z 176,A -41.0035,B 7.2093,C 0.3426,E1 7.3336,E2 492.8543} C_DIS
LIN {X 94.464,Y -94.8073,Z 176,A -42.8307,B 7.2091,C 0.3468,E1 7.33,E2 494.6857} C_DIS
LIN {X 91.0979,Y -98.046,Z 176,A -44.5526,B 7.2091,C 0.346,E1 7.3266,E2 496.3749} C_DIS
LIN {X 88.4734,Y -100.4208,Z 176,A -46.2579,B 7.2088,C 0.3524,E1 7.323,E2 498.1052} C_DIS
LIN {X 85.1056,Y -103.2907,Z 176,A -47.8963,B 7.2088,C 0.3516,E1 7.3196,E2 499.7136} C_DIS
LIN {X 80.1349,Y -107.1928,Z 176,A -50.6492,B 7.2085,C 0.3574,E1 7.3135,E2 502.475} C_DIS
LIN {X 76.7153,Y -109.6664,Z 176,A -52.5926,B 7.2083,C 0.363,E1 7.3091,E2 504.4369} C_DIS
LIN {X 73.1406,Y -112.082,Z 176,A -54.414,B 7.2081,C 0.3656,E1 7.3048,E2 506.2567} C_DIS
LIN {X 70.368,Y -113.8435,Z 176,A -56.2052,B 7.2077,C 0.3745,E1 7.3005,E2 508.0967} C_DIS
LIN {X 66.7319,Y -116.0121,Z 176,A -57.976,B 7.2076,C 0.3766,E1 7.2962,E2 509.8639} C_DIS
LIN {X 63.1387,Y -118.0059,Z 176,A -59.3835,B 7.2078,C 0.3732,E1 7.2928,E2 511.2293} C_DIS
LIN {X 58.3656,Y -120.438,Z 176,A -61.6587,B 7.2076,C 0.376,E1 7.2871,E2 513.5041} C_DIS
LIN {X 54.8454,Y -122.0792,Z 176,A -63.2203,B 7.2076,C 0.3765,E1 7.2832,E2 515.0544} C_DIS
LIN {X 51.7636,Y -123.4175,Z 176,A -64.5172,B 7.2076,C 0.3759,E1 7.2799,E2 516.3348} C_DIS
LIN {X 48.7272,Y -124.6477,Z 176,A -66.0373,B 7.2074,C 0.3795,E1 7.2759,E2 517.8706} C_DIS
LIN {X 45.5621,Y -125.839,Z 176,A -67.492,B 7.2074,C 0.3812,E1 7.2721,E2 519.3272} C_DIS
LIN {X 41.9569,Y -127.0869,Z 176,A -69.135,B 7.2072,C 0.383,E1 7.2677,E2 520.9726} C_DIS
LIN {X 38.0174,Y -128.3207,Z 176,A -70.8325,B 7.2072,C 0.3836,E1 7.2632,E2 522.6627} C_DIS
LIN {X 34.6034,Y -129.2825,Z 176,A -72.3062,B 7.2072,C 0.3842,E1 7.2593,E2 524.1318} C_DIS
LIN {X 31.0908,Y -130.1722,Z 176,A -73.9205,B 7.2071,C 0.3864,E1 7.2549,E2 525.7549} C_DIS
LIN {X 27.0464,Y -131.0725,Z 176,A -75.6126,B 7.2071,C 0.3864,E1 7.2503,E2 527.4381} C_DIS
LIN {X 23.386,Y -131.7745,Z 176,A -77.2237,B 7.207,C 0.3877,E1 7.2458,E2 529.052} C_DIS
LIN {X 19.3252,Y -132.4315,Z 176,A -79.0328,B 7.2069,C 0.3894,E1 7.2408,E2 530.8682} C_DIS
LIN {X 15.594,Y -132.9222,Z 176,A -80.5864,B 7.2069,C 0.3893,E1 7.2365,E2 532.4156} C_DIS
LIN {X 11.3082,Y -133.355,Z 176,A -82.4734,B 7.2069,C 0.3907,E1 7.2313,E2 534.3089} C_DIS
LIN {X 6.2467,Y -133.6886,Z 176,A -84.5559,B 7.2069,C 0.3899,E1 7.2255,E2 536.3815} C_DIS
LIN {X 2.7085,Y -133.8072,Z 176,A -86.1519,B 7.2068,C 0.3915,E1 7.221,E2 537.9883} C_DIS
LIN {X 2.7085,Y -133.8072,Z 176,A -86.1519,B 7.2068,C 0.3915,E1 7.221,E2 537.9883} C_DIS
Enddeposition()
LIN {X 0.9842,Y -134.7334,Z 176,A -86.2865,B 7.2069,C 0.3862,E1 7.2206,E2 538.0807} C_DIS
Startdeposition()
$VEL.CP = VEL_PRINT
LIN {X 4.41,Y -134.6688,Z 176,A -84.2149,B 7.2075,C 0.376,E1 7.2266,E2 535.9304} C_DIS
LIN {X 8.6287,Y -134.4632,Z 176,A -82.8875,B 7.2071,C 0.3831,E1 7.2302,E2 534.6618} C_DIS
LIN {X 14.2296,Y -133.9859,Z 176,A -80.5093,B 7.2071,C 0.3824,E1 7.2368,E2 532.2839} C_DIS
LIN {X 17.7519,Y -133.5649,Z 176,A -79.0343,B 7.2071,C 0.3822,E1 7.2408,E2 530.8122} C_DIS
LIN {X 21.3828,Y -133.0339,Z 176,A -77.2377,B 7.2074,C 0.3774,E1 7.2459,E2 528.9848} C_DIS
LIN {X 25.9662,Y -132.2152,Z 176,A -75.5232,B 7.2072,C 0.3805,E1 7.2505,E2 527.3028} C_DIS
LIN {X 29.6406,Y -131.4389,Z 176,A -73.8779,B 7.2073,C 0.3786,E1 7.255,E2 525.6502} C_DIS
LIN {X 33.1023,Y -130.6095,Z 176,A -72.3846,B 7.2073,C 0.3777,E1 7.2591,E2 524.1585} C_DIS
LIN {X 36.4825,Y -129.7061,Z 176,A -70.9334,B 7.2074,C 0.377,E1 7.263,E2 522.711} C_DIS
LIN {X 39.7287,Y -128.749,Z 176,A -69.5137,B 7.2074,C 0.376,E1 7.2667,E2 521.2927} C_DIS
LIN {X 42.7292,Y -127.7843,Z 176,A -68.1983,B 7.2075,C 0.375,E1 7.2702,E2 519.9795} C_DIS
LIN {X 45.9053,Y -126.678,Z 176,A -66.7766,B 7.2075,C 0.3737,E1 7.274,E2 518.5578} C_DIS
LIN {X 49.0778,Y -125.4831,Z 176,A -65.3311,B 7.2077,C 0.3719,E1 7.2777,E2 517.1107} C_DIS
LIN {X 52.2142,Y -124.2109,Z 176,A -63.8859,B 7.2077,C 0.3701,E1 7.2815,E2 515.6637} C_DIS
LIN {X 55.2603,Y -122.8858,Z 176,A -62.4644,B 7.2079,C 0.3682,E1 7.2851,E2 514.24} C_DIS
LIN {X 59.0476,Y -121.1128,Z 176,A -60.8125,B 7.2079,C 0.368,E1 7.2892,E2 512.6028} C_DIS
LIN {X 61.4554,Y -119.9079,Z 176,A -59.6088,B 7.2079,C 0.3653,E1 7.2923,E2 511.3906} C_DIS
LIN {X 65.4026,Y -117.8029,Z 176,A -56.952,B 7.2088,C 0.3493,E1 7.299,E2 508.6361} C_DIS
LIN {X 70.4034,Y -114.8845,Z 176,A -55.1822,B 7.2084,C 0.3576,E1 7.303,E2 506.9527} C_DIS
LIN {X 73.5816,Y -112.8756,Z 176,A -53.6072,B 7.2084,C 0.3554,E1 7.3067,E2 505.3793} C_DIS
LIN {X 77.2601,Y -110.3906,Z 176,A -51.7016,B 7.2087,C 0.3518,E1 7.3111,E2 503.4698} C_DIS
LIN {X 80.6417,Y -107.9447,Z 176,A -49.7976,B 7.2089,C 0.3463,E1 7.3154,E2 501.5478} C_DIS
LIN {X 85.2108,Y -104.3754,Z 176,A -47.5663,B 7.2089,C 0.3459,E1 7.3202,E2 499.344} C_DIS
LIN {X 88.4453,Y -101.6491,Z 176,A -45.4561,B 7.2094,C 0.3368,E1 7.3248,E2 497.1926} C_DIS
LIN {X 91.3781,Y -99.0212,Z 176,A -44.233,B 7.2092,C 0.3416,E1 7.3272,E2 496.0253} C_DIS
LIN {X 94.1143,Y -96.4246,Z 176,A -42.5351,B 7.2094,C 0.3365,E1 7.3306,E2 494.314} C_DIS
LIN {X 97.233,Y -93.2785,Z 176,A -40.6681,B 7.2096,C 0.3328,E1 7.3343,E2 492.4474} C_DIS
LIN {X 100.2465,Y -90.032,Z 176,A -38.8157,B 7.2097,C 0.3293,E1 7.3378,E2 490.5972} C_DIS
LIN {X 103.2285,Y -86.5965,Z 176,A -36.9294,B 7.2099,C 0.3258,E1 7.3412,E2 488.7151} C_DIS
LIN {X 106.1542,Y -82.9847,Z 176,A -34.9501,B 7.2101,C 0.3212,E1 7.3446,E2 486.7337} C_DIS
LIN {X 108.5502,Y -79.8245,Z 176,A -33.2491,B 7.2103,C 0.3169,E1 7.3474,E2 485.0292} C_DIS
LIN {X 111.7434,Y -75.29,Z 176,A -31.2616,B 7.2103,C 0.3181,E1 7.3505,E2 483.0862} C_DIS
LIN {X 113.3072,Y -72.9155,Z 176,A -29.7197,B 7.2106,C 0.3089,E1 7.353,E2 481.5012} C_DIS
LIN {X 115.7159,Y -69.0284,Z 176,A -27.9717,B 7.2106,C 0.3077,E1 7.3555,E2 479.776} C_DIS
LIN {X 118.5532,Y -64.0337,Z 176,A -25.4925,B 7.211,C 0.3008,E1 7.3588,E2 477.2899} C_DIS
LIN {X 120.4085,Y -60.4721,Z 176,A -23.6496,B 7.2113,C 0.2938,E1 7.3612,E2 475.4283} C_DIS
LIN {X 122.6225,Y -55.8453,Z 176,A -21.6817,B 7.2113,C 0.292,E1 7.3635,E2 473.4851} C_DIS
LIN {X 124.0186,Y -52.6745,Z 176,A -20.3519,B 7.2113,C 0.2908,E1 7.3649,E2 472.1721} C_DIS
LIN {X 125.0792,Y -50.0982,Z 176,A -19.1759,B 7.2115,C 0.2877,E1 7.3662,E2 470.9959} C_DIS
LIN {X 126.2595,Y -47.0442,Z 176,A -17.8013,B 7.2116,C 0.2843,E1 7.3675,E2 469.6223} C_DIS
LIN {X 127.5936,Y -43.3018,Z 176,A -16.1807,B 7.2118,C 0.2809,E1 7.369,E2 468.0087} C_DIS
LIN {X 128.4419,Y -40.7107,Z 176,A -15.0386,B 7.2118,C 0.2781,E1 7.37,E2 466.8676} C_DIS
LIN {X 129.4112,Y -37.5163,Z 176,A -13.0049,B 7.2125,C 0.2626,E1 7.3716,E2 464.7552} C_DIS
LIN {X 130.733,Y -32.6158,Z 176,A -11.5403,B 7.2122,C 0.2696,E1 7.3726,E2 463.376} C_DIS
LIN {X 131.3216,Y -30.1544,Z 176,A -10.4882,B 7.2122,C 0.267,E1 7.3732,E2 462.3259} C_DIS
LIN {X 132.0101,Y -26.9811,Z 176,A -9.0517,B 7.2125,C 0.262,E1 7.3741,E2 460.8812} C_DIS
LIN {X 132.7863,Y -22.8675,Z 176,A -7.1949,B 7.2127,C 0.2555,E1 7.375,E2 459.0131} C_DIS
LIN {X 133.4157,Y -18.8402,Z 176,A -5.5922,B 7.2127,C 0.253,E1 7.3756,E2 457.4252} C_DIS
LIN {X 133.9471,Y -14.5896,Z 176,A -3.8569,B 7.2129,C 0.2494,E1 7.3762,E2 455.6991} C_DIS
LIN {X 134.3099,Y -10.764,Z 176,A -1.5165,B 7.2135,C 0.2314,E1 7.3768,E2 453.2685} C_DIS
LIN {X 134.644,Y -5.0709,Z 176,A 0.1977,B 7.2133,C 0.2379,E1 7.3769,E2 451.6416} C_DIS
LIN {X 134.7384,Y -0.7211,Z 176,A 1.9266,B 7.2134,C 0.2348,E1 7.377,E2 449.9263} C_DIS
LIN {X 134.7116,Y 2.7924,Z 176,A 3.5184,B 7.2136,C 0.2287,E1 7.377,E2 448.3211} C_DIS
LIN {X 134.46,Y 8.6795,Z 176,A 5.7352,B 7.2136,C 0.2269,E1 7.3766,E2 446.1382} C_DIS
LIN {X 134.2502,Y 11.4709,Z 176,A 7.0332,B 7.2138,C 0.2215,E1 7.3763,E2 444.8258} C_DIS
LIN {X 133.8665,Y 15.324,Z 176,A 8.6978,B 7.214,C 0.2165,E1 7.3758,E2 443.1577} C_DIS
LIN {X 133.3504,Y 19.2972,Z 176,A 10.3122,B 7.214,C 0.2133,E1 7.3752,E2 441.5531} C_DIS
LIN {X 132.6904,Y 23.4094,Z 176,A 12.0571,B 7.2142,C 0.2088,E1 7.3744,E2 439.8101} C_DIS
LIN {X 132.0049,Y 27.0064,Z 176,A 13.5811,B 7.2143,C 0.205,E1 7.3736,E2 438.289} C_DIS
LIN {X 131.1837,Y 30.7578,Z 176,A 15.3175,B 7.2145,C 0.1985,E1 7.3725,E2 436.5387} C_DIS
LIN {X 130.1632,Y 34.816,Z 176,A 16.8955,B 7.2145,C 0.1973,E1 7.3714,E2 434.9843} C_DIS
LIN {X 129.2969,Y 37.9066,Z 176,A 18.2292,B 7.2146,C 0.1941,E1 7.3704,E2 433.6535} C_DIS
LIN {X 128.2586,Y 41.2846,Z 176,A 19.7389,B 7.2147,C 0.1899,E1 7.3691,E2 432.142} C_DIS
LIN {X 126.8695,Y 45.3742,Z 176,A 22.1073,B 7.2151,C 0.1751,E1 7.3669,E2 429.7064} C_DIS
LIN {X 125.1428,Y 49.9404,Z 176,A 23.4168,B 7.2149,C 0.1837,E1 7.3656,E2 428.4906} C_DIS
LIN {X 124.121,Y 52.4293,Z 176,A 24.6386,B 7.2149,C 0.1793,E1 7.3643,E2 427.2586} C_DIS
LIN {X 122.9083,Y 55.2101,Z 176,A 25.9587,B 7.2151,C 0.1753,E1 7.3628,E2 425.934} C_DIS
LIN {X 121.5322,Y 58.1763,Z 176,A 27.3404,B 7.2151,C 0.1719,E1 7.3612,E2 424.5525} C_DIS
LIN {X 119.7046,Y 61.8547,Z 176,A 29.1029,B 7.2153,C 0.1672,E1 7.3589,E2 422.7873} C_DIS
LIN {X 117.6644,Y 65.6532,Z 176,A 30.9569,B 7.2153,C 0.1622,E1 7.3564,E2 420.9299} C_DIS
LIN {X 115.4083,Y 69.5417,Z 176,A 32.7987,B 7.2155,C 0.1588,E1 7.3538,E2 419.0957} C_DIS
LIN {X 113.1437,Y 73.1686,Z 176,A 34.6052,B 7.2155,C 0.1546,E1 7.3511,E2 417.2898} C_DIS
LIN {X 110.671,Y 76.8572,Z 176,A 36.433,B 7.2156,C 0.1512,E1 7.3482,E2 415.4686} C_DIS
LIN {X 108.4811,Y 79.9185,Z 176,A 38.0011,B 7.2156,C 0.1481,E1 7.3457,E2 413.9038} C_DIS
LIN {X 104.6308,Y 84.8961,Z 176,A 40.7277,B 7.2158,C 0.1412,E1 7.341,E2 411.1699} C_DIS
LIN {X 101.6129,Y 88.4869,Z 176,A 42.6291,B 7.2158,C 0.1385,E1 7.3375,E2 409.2794} C_DIS
LIN {X 98.6504,Y 91.778,Z 176,A 44.8429,B 7.2161,C 0.1287,E1 7.3333,E2 407.0243} C_DIS
LIN {X 95.7578,Y 94.7924,Z 176,A 46.2407,B 7.2161,C 0.1318,E1 7.3306,E2 405.6726} C_DIS
LIN {X 92.6164,Y 97.8638,Z 176,A 48.3576,B 7.2161,C 0.1237,E1 7.3263,E2 403.5246} C_DIS
LIN {X 89.8738,Y 100.3882,Z 176,A 49.6054,B 7.2161,C 0.1266,E1 7.3238,E2 402.3179} C_DIS
LIN {X 86.5957,Y 103.2292,Z 176,A 51.4387,B 7.2161,C 0.1233,E1 7.3199,E2 400.4856} C_DIS
LIN {X 83.0819,Y 106.0779,Z 176,A 53.3481,B 7.2162,C 0.1201,E1 7.3157,E2 398.5776} C_DIS
LIN {X 79.7303,Y 108.6193,Z 176,A 55.1192,B 7.2162,C 0.1174,E1 7.3117,E2 396.8083} C_DIS
LIN {X 75.1805,Y 111.8162,Z 176,A 57.4069,B 7.2162,C 0.1148,E1 7.3065,E2 394.5297} C_DIS
LIN {X 71.7339,Y 114.0587,Z 176,A 59.1811,B 7.2163,C 0.1117,E1 7.3023,E2 392.7524} C_DIS
LIN {X 67.9759,Y 116.3377,Z 176,A 60.9931,B 7.2163,C 0.1099,E1 7.298,E2 390.9472} C_DIS
LIN {X 64.1809,Y 118.4739,Z 176,A 62.8871,B 7.2164,C 0.1066,E1 7.2933,E2 389.0481} C_DIS
LIN {X 60.4974,Y 120.3956,Z 176,A 64.5117,B 7.2164,C 0.1067,E1 7.2893,E2 387.4408} C_DIS
LIN {X 57.8745,Y 121.6764,Z 176,A 65.7742,B 7.2164,C 0.1048,E1 7.2862,E2 386.1757} C_DIS
LIN {X 54.6964,Y 123.138,Z 176,A 67.2332,B 7.2164,C 0.1035,E1 7.2825,E2 384.7202} C_DIS
LIN {X 51.3565,Y 124.569,Z 176,A 69.0327,B 7.2165,C 0.0976,E1 7.2777,E2 382.89} C_DIS
Enddeposition()
END
